(* CODESYS project Base (4).library
   Company: Photara
   DefaultNamespace: Base
   Title: Base
   Placeholder: Base
   Author: Scott Kinder
   Version: 2025.10.17.4

Project tree, tasks and I/O mapping:
  libraries: Tc2_EtherCAT, * (Beckhoff Automation GmbH); Tc2_Standard, * (Beckhoff Automation GmbH); Tc2_System, * (Beckhoff Automation GmbH); Tc2_Utilities, * (Beckhoff Automation GmbH); Tc3_EventLogger, * (Beckhoff Automation GmbH); Tc3_JsonXml, * (Beckhoff Automation GmbH); TcUnit, 1.3.1 (www.tcunit.org)
  Base/
    POUs/
      function block FB_BaseCyclic [ST]: _ConfigurationCyclic, _UpdateStatusEdgeTracking, CyclicLogic, Initialized
      function block FB_BaseStatic [ST]: Busy, Error, ErrorID, Initialize, P_BaseConfiguration, P_BaseStatus, TraceWithSeverity, _FormatLogEntry, _Initialize, _InitializeChildrenDependencies, _InitializeReferences, _SetDependencyConfiguration, RaiseAlarm
    global variables GC_Base
    global variables GPL_Base
    interface I_BaseCyclic: CyclicLogic, Initialized
    interface I_BaseStatic: Busy, Error, ErrorID, Initialize, P_BaseConfiguration, P_BaseStatus, TraceWithSeverity
  Command/
    ITFs/
      interface I_Command: Abort, Cancel, Complete, Execute, InjectConfigurations, P_CommandStatus, Pause, Queue, Reset, Resume, Validate
      interface I_CommandConfiguration: P_CommandConfiguration
      interface I_TestClock: SetElapsedTime
      interface I_Timer: P_ElapsedTime, P_IsElapsed, ResetTimer, StartTimer, StopTimer
    POUs/
      function block FB_Command [ST]: Abort, Cancel, Complete, Execute, InjectConfigurations, P_CommandStatus, Pause, Queue, Reset, Resume, Validate, _Initialize, _InitializeChildrenDependencies, _InitializeReferences, _SetDependencyConfiguration, _AbortCommand, _AbortCommandInterlockLost, _ConfigurationCyclic, _EvaluateConfiguration, _FormatResultString, _FormatStepStateString, _HandleAutoReset, _LogCommand, _MonitorInterlocks, _ProcessStateTransitions, _ResetCommand, _ResolveCommandConfiguration, _ResolveCommandStatus, _ResolvePermIntlkConfiguration, _UpdateComponentStatus, _UpdateStatusEdgeTracking, _ValidateCommand, CyclicLogic, P_CommandConfiguration, P_PermIntlkConfiguration
      function block FB_CommandElapsedTimer [ST]: P_ElapsedTime, P_IsElapsed, ResetTimer, StartTimer, StopTimer, CyclicLogic, InjectConfiguration
  Component/
    GVLs/
      global variables GC_Component
      global variables GPL_Component
    ITFs/
      interface I_ComponentBase: InjectSystemInterfaces, Reset
      interface I_ComponentFull: DequeueCommand, EnqueueCommand, ExecuteCommand, GetIndexByPOUName, HMICommunication, InjectCommandQueue, P_CommandQueue, P_ComponentConfiguration, P_ComponentStatus, ResetAllCommands
    POUs/
      function block FB_Component [ST]: DequeueCommand, EnqueueCommand, ExecuteCommand, GetIndexByPOUName, HMICommunication, InjectCommandQueue, P_CommandQueue, P_ComponentConfiguration, P_ComponentStatus, Reset, ResetAllCommands, _Initialize, _InitializeChildrenDependencies, _InitializeReferences, _SetCommandIndices, _SetCommandPermIntlkConfiguration, FB_Init, InjectCommandConfiguration, InjectPermIntlkConfiguration, InjectSystemInterfaces, _BuildTables, _ClearTempCmdObj, _CommandsCyclic, _ComponentCyclic, _DequeueCommand, _DispatchValid, _EnqueueCommand, _EvaluateCompletionConditions, _InjectCommandConfiguration, _InjectPermIntlkConfiguration, _ObtainAmsNetId, _ProcessCommandQueue, _TryRehashDispatchIndex, _UpdateBusyStatus, _UpdateComponentStatus, CyclicLogic
  Configuration/
    function block FB_CmdPermIntlkConfiguration [ST]: _InitializeReferences, P_CommandConfiguration, P_PermIntlkConfiguration
  ControlMode/
    GVLs/
      global variables GC_ControlMode
      global variables GPL_ControlMode
    ITFs/
      interface I_ControlMode: ChangeMode, P_ControlMode
    POUs/
      function block FB_ControlMode [ST]: ChangeMode, P_ControlMode, _EvaluateCompletionConditions, _UpdateComponentStatus, InjectControlModeCmdPermIntlkConfigurations
  Debounce/
    function block FB_Debounce [ST]: _InitializeReferences, CyclicLogic, P_DebounceConfiguration, P_DebounceStatus, P_RawSignal
    interface I_Debounce: P_DebounceStatus, P_RawSignal
    interface I_DebounceConfiguration: P_DebounceConfiguration
  DUTs/
    Base/
      data type E_DataType
      data type E_HttpStatusCode
      data type E_LinkStatus
      data type ST_BaseConfiguration
      data type ST_BaseStatus
      data type ST_BitSignal
      data type ST_OpStatus
      data type ST_Parameter
      data type ST_PlcSystem
    Command/
      data type E_CommandPriority
      data type E_CommandResult
      data type E_CommandState
      data type ST_CommandConfiguration
      data type ST_CommandStatus
    Component/
      data type E_ComponentTriggerMode
      data type ST_ComponentCommand
      data type ST_ComponentConfiguration
      data type ST_ComponentStatus
    Configuration/
      data type E_ConfigurationResolution
    Debounce/
      data type ST_DebounceConfiguration
      data type ST_DebounceStatus
    EtherCAT/
      data type ST_EtherCATAdsAddr
      data type ST_EtherCATInfoData
      data type ST_EtherCATStatus
      data type ST_EtherCATWcState
    EventHandling/
      data type ST_EventLogHandlerConfiguration
      data type ST_EventLogHandlerStatus
      data type ST_PersistentStorageStatus
    File/
      Structs/
        data type ST_AmsNetId
        data type ST_FileHandlerBaseStatus
        data type ST_FileHandlerConfiguration
        data type ST_FileHandlerCSVConfiguration
        data type ST_FileHandlerCSVStatus
        data type ST_FileHandlerJsonStatus
        data type ST_FileOpStatus
      data type E_FileFormat
    Hash/
      data type ST_HashTableConfiguration
      data type ST_HashTableStatus
    LogTrace/
      data type E_LogTraceWhen
      data type ST_LogBackoffState
      data type ST_LogMetrics
      data type ST_LogTraceConfiguration
      data type ST_LogTraceStatus
      data type ST_LogTraceWhat
    PermIntlk/
      data type E_ModePermIntlk
      data type ST_PermIntlkConfiguration
      data type ST_PermIntlkConfigurationCondition
      data type ST_PermIntlkStatus
      data type ST_PermIntlkStatusCondition
    RingBuffer/
      data type ST_LogEntry
      data type ST_RingBufferCfg
      data type ST_RingBufferStatus
      data type ST_SystimeICmd
      data type ST_SystimeString
    Safety/
      data type ST_SafetyGroupConfiguration
      data type ST_SafetyGroupStatus
    Sequencer/
      data type E_Operation
      data type E_PackMLState
      data type ST_Operation
      data type ST_OperationSequencerConfiguration
      data type ST_OperationSequencerStatus
      data type ST_PackMLSequencerConfiguration
      data type ST_PackMLSequencerStatus
  EventHandling/
    ITFs/
      interface I_LogHandler: AddToEventLog, LogDequeue, MonitorPlcSystem, P_EventLogHandlerStatus
      interface I_LogHandlerConfiguration: P_EventLogHandlerConfiguration
      interface I_PersistentStorage: AddEntry, P_MessagesSentThisScan
      interface I_TraceEvent: AddContext, SetMessage, SetSeverity
    function block FB_EventLogHandler [ST]: CyclicLogic, AddToEventLog, LogDequeue, MonitorPlcSystem, P_EventLogHandlerStatus, P_EventLogHandlerConfiguration, _InitializeChildrenDependencies, _InitializeReferences, _ProcessLogEntry, _UpdatePerformanceMetrics, _UpdateSeverityMetrics, CalculateDynamicRate, HandlePersistenceFailure, UpdateBufferHealthMetrics
    function block FB_PersistentEventLog [ST]: _InitializeChildrenDependencies, _InitializeReferences, AddEntry, P_MessagesSentThisScan
    function block FB_TraceEvent [ST]: AddContext, SetMessage, SetSeverity
    function block FB_UniversalAlarm [ST]: AddContext, Clear, Confirm, Raise, SetMessage, SetSeverity
    function block FB_UniversalMessage [ST]: AddContext, Send, SetMessage, SetSeverity
    global variables GVL_System
  File/
    Function Blocks/
      function block FB_FileHandlerBase [ST]: P_FileHandlerBaseConfiguration, _InitializeReferences, CyclicLogic, P_FileHandlerBaseStatus
      function block FB_FileHandlerJson [ST]: CyclicLogic
    Interfaces/
      interface I_FileHandlerBase: AppendToFileByPointer, CloseFile, CreateFile, DeleteFile, OpenFile, ReadFromFile, RenameFile, WriteFile, P_FileHandlerBaseStatus
      interface I_FileHandlerBaseConfiguration: P_FileHandlerBaseConfiguration
      interface I_FileHandlerCsv: AppendToFileByString, AppendToFileBySystimeString, P_AppendRingBufferStatus, P_FileHandlerCsvStatus
      interface I_FileHandlerJson
    global variables GC_File
    global variables GPL_File
  Functions/
    Numbers/
      function F_IsPowerOfTwo_UINT [ST]
      function F_MapLREAL [ST]
    Strings/
      function F_GetAllButFirstWord [ST]
      function F_GetFirstWordInString [ST]
      function F_GetLastWordInString [ST]
      function F_ReplaceInString [ST]
      function F_TrimString [ST]
    Time/
      function F_DateTimeConvertedAsT_MaxString [ST]
      function F_FILETIME64_TO_LTIME [ST]
      function F_FileTimeToString [ST]
      function F_SystemTimeUtcCorrected [ST]
  Hashing/
    ITFs/
      interface I_HashFunction: Hash
      interface I_HashTableBase: Clear, GetIndex, Insert, P_HashTableStatus
      interface I_HashTableConfiguration: P_HashTableConfiguration
      interface I_HashTableExt: Contains, LoadFactorExceeded, Rehash, Remove
    POUs/
      function block FB_Hash_djb2 [ST]: Hash, P_TP_HashTableStatus
      function block FB_HashTable [ST]: Clear, GetIndex, Insert, P_HashTableStatus, P_HashTableConfiguration, _Initialize, _InitializeChildrenDependencies, _InitializeHashTable, _InitializeReferences, InjectHashFunction
    global variables GPL_HashTable
  PermIntlk/
    GVLs/
      global variables GC_PermIntlk
      global variables GPL_PermIntlk
    ITFs/
      interface I_PermIntlk: Evaluate, InjectPermIntlkConfiguration, P_OK, P_PermIntlkStatus
      interface I_PermIntlkConfiguration: P_PermIntlkConfiguration
    POUs/
      function block FB_PermIntlk [ST]: Evaluate, P_OK, P_PermIntlkConfiguration, _Initialize, _InitializeReferences, _SetElementIndices, _EvaluateConfiguration, _EvaluateOK, _LogMessage, _PermMsgIndexForMessage, _ResolvePermIntlkConfiguration, _ResolvePermIntlkStatus, _ConfigurationCyclic, CyclicLogic, InjectPermIntlkConfiguration, P_PermIntlkStatus, ReinitObjects
      function block FB_PermIntlkCommand [ST]: CyclicLogic, InjectCommandConfiguration
  PRGs/
    program PRG_LOG [ST]
    program PRG_PRETEST [ST]
    program PRG_TEST [ST]
  RingBuffer/
    GVLs/
      global variables GPL_RingBuffer
    ITFs/
      interface I_RingBufferBase: ClearLastRemoved, ClearStatusFlagAdded, ClearStatusFlagPeeked, ClearStatusFlagRead, ClearStatusFlagRemoved, P_ObjectWasAdded, P_ObjectWasPeeked, P_ObjectWasRead, P_ObjectWasRemoved, P_RingBufferStatus, RemoveObject
      interface I_RingBufferICmd: AddObject, P_Buffer, P_LastObjectPeeked, P_LastObjectRead, P_LastObjectRemoved, PeekObject, ReadObject
      interface I_RingBufferKeyString: AddObject, P_Buffer, P_LastObjectPeeked, P_LastObjectRead, P_LastObjectRemoved, PeekObject, ReadObject
      interface I_RingBufferLogEntry: AddObject, P_Buffer, P_LastObjectPeeked, P_LastObjectRead, P_LastObjectRemoved, PeekObject, ReadObject
      interface I_RingBufferString: AddObject, P_Buffer, P_LastObjectPeeked, P_LastObjectRead, P_LastObjectRemoved, PeekObject, ReadObject
      interface I_RingBufferUINT: AddObject, P_Buffer, P_LastObjectPeeked, P_LastObjectRead, P_LastObjectRemoved, PeekObject, ReadObject
    POUs/
      function block FB_RingBufferBase [ST]: _Initialize, _InitializeReferences, UpdateObjectCtInBuffers, P_ObjCountInBuffer, P_ObjectWasAdded, P_ObjectWasPeeked, P_ObjectWasRead, P_ObjectWasRemoved, ClearLastRemoved, IncrementPointer, UpdateRemovePointer, UpdateWritePointer, ClearStatusFlagAdded, ClearStatusFlagPeeked, ClearStatusFlagRead, ClearStatusFlagRemoved, ClearStatusFlags, WrapPointer
      function block FB_RingBufferICmd [ST]: ClearLastRemoved, P_RingBufferStatus, RemoveObject, AddObject, P_Buffer, P_LastObjectPeeked, P_LastObjectRead, P_LastObjectRemoved, PeekObject, ReadObject, UpdateRemovePointer, UpdateWritePointer, _Initialize, ClearBuffer
      function block FB_RingBufferKeyString [ST]: AddObject, ClearLastRemoved, P_LastObjectPeeked, P_LastObjectRead, P_LastObjectRemoved, P_RingBufferStatus, PeekObject, ReadObject, RemoveObject, UpdateRemovePointer, UpdateWritePointer, _Initialize, ClearBuffer, P_Buffer
      function block FB_RingBufferLogEntry [ST]: AddObject, ClearLastRemoved, P_LastObjectPeeked, P_LastObjectRead, P_LastObjectRemoved, P_RingBufferStatus, PeekObject, ReadObject, RemoveObject, UpdateRemovePointer, UpdateWritePointer, _Initialize, ClearBuffer, P_Buffer
      function block FB_RingBufferString [ST]: ClearLastRemoved, P_RingBufferStatus, RemoveObject, AddObject, P_LastObjectPeeked, P_LastObjectRead, P_LastObjectRemoved, PeekObject, ReadObject, UpdateRemovePointer, UpdateWritePointer, _Initialize, ClearBuffer, P_Buffer
      function block FB_RingBufferUINT [ST]: ClearLastRemoved, P_RingBufferStatus, RemoveObject, AddObject, P_LastObjectPeeked, P_LastObjectRead, P_LastObjectRemoved, PeekObject, ReadObject, UpdateRemovePointer, UpdateWritePointer, _Initialize, ClearBuffer, P_Buffer
  Safety/
    GVLs/
      global variables GC_Safety
      global variables GPL_Safety
    function block FB_SafetyDevice [ST]: CyclicLogic
    function block FB_SafetyGroup [ST]: _InitializeReferences, CyclicLogic, P_SafetyGroupConfiguration, P_SafetyGroupStatus, Reset
  Tests/
    FB_CommandConfigured/
      function block FB_CommandConfigured [ST]
    MockFBs/
      function block FB_CommandUnderTest [ST]: SetCommandConfiguration, SetCommandStatus
      function block FB_ComponentDerivative [ST]: P_TP_iSystemPermIntlk, _EvaluateCompletionConditions, _UpdateComponentStatus
      function block FB_ImplBaseCyclic [ST]
      function block FB_ImplBaseStatic [ST]
    TestFunctions/
      function GivenValidCommand [ST]
      function ThenAssertState [ST]
      function WhenExecuteCommand [ST]
    TestInterfaces/
      interface I_CommandUnderTest: SetCommandStatus
    function block FB_BaseCyclicTests [ST]: GivenCyclicCallInitCompleteOK, GivenNoCyclicCallInitCompleteNOK
    function block FB_BaseStaticTests [ST]: GivenInitializationConfigurationReferenceOK, GivenNoInitializationConfigurationReferenceNOK
    function block FB_CommandTestsI [ST]: GivenCommand_WhenCancelCalledIfCommandNotAlreadyDequeuedExpectCommandRemovedFromQueue, GivenCommand_WhenExecuteCalled_ExpectExecutionOccurs, GivenCommand_WhenQueueCalledExpectCommandAddedToQueue, GivenCommand_WhenResetCalled_ExpectStateCleared, GivenCommandInIdleState_WhenCancel_ExpectNoActionTaken, GivenCommandPaused_WhenAbort_ExpectCommandAbortedAndStatusUpdated, GivenCommandQueued_WhenAbort_ExpectCommandAbortedAndStatusUpdated, GivenCommandQueued_WhenCancel_ExpectCommandRemovedFromQueue, GivenComponentReset_WhenResetCalled_ExpectAllCommandStateCleared, TEST_AbortAfterComplete_StatePreservation, TEST_Cancel_FromQueuedState, TEST_Execute_StateMachineProgression, TEST_Execute_TransitionsFromAcceptedToOk, TEST_Reset_ClearsCommandState, TEST_CommandAttemptsExceedRetryCount_ResultTooManyRequests, TEST_CommandTimeout_TriggersReset, TEST_PermIntlkLostDuringBusy_CommandAbortedWithInterlockLost, GivenCommandAlreadyRunning_WhenExecute_ExpectConflictResult, TEST_CommandCompletes_StatusDoneAndBusyCleared, TEST_CompleteState_PreservesAbortedResult, TEST_CompleteState_PreservesTimeoutResult, TEST_CompleteState_SetsOkForSuccessfulCompletion, TEST_Forbidden_ResumeWithoutPermissive_ReturnsForbidden, TEST_OperatorAbort_VsInterlockAbort_DifferentResults, TEST_TerminalResults_ErrorFlagConsistency, TEST_ValidationOK_InterlockDropDuringExecution, TEST_ValidCommand_ExpectExecuted, GivenCommand_WhenCyclicLogicCalled_ExpectStateUpdated, GivenCommand_WhenPauseCalledExpectCommandPauses, GivenCommand_WhenResumeCalledExpectCommandResumes, GivenCommandExecuted_WhenCyclicLogicRuns_ExpectStateProgression, GivenCommandPaused_WhenResume_ExpectCommandResumesExecution, GivenRunningCommand_WhenPause_ExpectCommandTransitionsToPausedState, GivenTimerStarted_WhenCyclicLogicRuns_ExpectElapsedTimeIncreases, GivenTimerStopped_WhenCyclicLogicRuns_ExpectElapsedTimeRemainsConstant, TEST_CyclicLogic_StateMachineProgression, TEST_EdgeTriggered_StateMachineExecution, TEST_PauseResume_StateTransitions, TEST_StepState_TransitionsAndValidation, GivenCommand_WhenValidateCalled_ExpectPermissiveOK, GivenCommand_WhenValidateCalled_ExpectValidationResultMatchesConfiguration, GivenCommandInvalid_WhenValidateCalled_ExpectFalse, GivenCommandValidated_WhenValidateCalled_ExpectTrue, GivenInjectedConfigurationsValid_WhenInjectConfigurations_ExpectInterfacesStoredAndInitialized, GivenInvalidConfiguration_WhenInjectConfigurationCalled_ExpectInitializationFailure, GivenInvalidConfigurations_WhenInjectConfigurations_ExpectInitializationFailure, GivenValidConfiguration_WhenInjectConfigurationCalled_ExpectConfigurationStored, TEST_ComponentBusyDuringValidation_ResultConflict, TEST_InjectConfigurations_StoresInterfacesProperly, TEST_InterfaceInjectionConfigurationResolution, TEST_PermissiveFalseDuringValidation_ResultForbidden, TEST_Validate_ReturnsProperResultBasedOnPermissives, TEST_Validate_WithContinuousEvaluation
    function block FB_CommandTestsII [ST]: TEST_Abort_AfterComplete_IgnoredWithWarning, TEST_Abort_WhenIdleQueued_SetsResultAbortedAndRemovesFromQueue, TEST_Cancel_WhenBusy_RejectedWithWarning_NoStateChange, TEST_Execute_HappyPath_TransitionsToMonitorAndCompletesOk, TEST_Execute_WhenPermissiveMissing_ReturnsForbidden, TEST_RetryCount_IncrementOnExecutionStartOnly, TEST_TimeoutAndInterlockLost_SameCycle_PrioritizeInterlockLost, TEST_Complete_Error_PersistsUntilReset, TEST_Complete_Ok_AutoResetsNextCycle, TEST_SystematicStateValidation_IdleStates, TEST_SystematicStateValidation_TerminalStates, TEST_Config_FallbackToLocal_WhenInjectedInvalid, TEST_Config_RecoveryToInjected_WhenValidAgain, TEST_Execute_ValidatesBeforeAccepting, TEST_RuntimeCommandConfigLoss_InjectedRefsInvalidatedDuringExecution, TEST_RuntimeCommandConfigRecovery_ValidRefsRestoredDuringExecution, TEST_AbortDuringCompletionWait, TEST_CompletionCallbackToSequencer, TEST_CompletionConditionEvaluation, TEST_CompletionWithInterlockDrop, TEST_DiscreteCompletionCondition, TEST_DynamicCompletionConditionUpdate, TEST_FastCompletionInOneScan, TEST_MotionCompletionCondition, TEST_OperationToCommandTranslation, TEST_RecipeManagerProvidesCommandConfig, TEST_TimeBasedCompletionCondition
    function block FB_CommandTestsIII [ST]: TEST_MethodEnablement_BusyState_ShouldAllowAbortRejectExecute, TEST_MethodEnablement_DoneState_ShouldAllowResetRejectExecute, TEST_MethodEnablement_IdleWithInterlockOK_ShouldAllowExecute, TEST_MethodEnablement_IdleWithoutInterlockOK_ShouldRejectExecute, TEST_InterlockInvalidConfigurationDuringValidation_ReturnsBadRequest, TEST_InterlockReferenceLostDuringExecution_FallsBackOrAborts, TEST_InterlockDrop_AbortsCommandWhenConfigured, TEST_InterlockDrop_FromMonitorState_CommandAborted, TEST_InterlockLost_ComprehensiveStateTransitions, TEST_InterlockLost_FromExecuteState, TEST_InterlockLost_SetsCorrectResult, TEST_TimerCompletionTime_SetOnCommandComplete, TEST_TimerIntegration_WithCommandStateMachine, TEST_TimerPauseResume_ElapsedTimeAccuracy, TEST_TimerStopsOnCommandComplete_NotTimeout, TEST_TimerTriggerTime_SetOnCommandStart
    function block FB_CommandTestsIV [ST]: TEST_Abort_ErrorClassification, TEST_Cancel_RemovesCommandFromQueue, TEST_Cancel_SetsCommandStatusToCancelled, TEST_Cancel_SetsResultToCancelled, TEST_BadRequest_InterlockMisconfigured_ReturnsBadRequest, TEST_BusyCommandElapsedTimeEqualsTimeout_CommandAborted, TEST_AcceptedCommand_WhenExecuted_ResultBecomesOk, TEST_Command_LocalReferences_InitializedProperly, TEST_Command_MissingConfigInterface_FallbackToLocal, TEST_Command_PermIntlkChild_Initialized, TEST_CommandStatus_ConfigRef_PointsToConfiguration
    function block FB_CommandTestsV [ST]: TEST_ConfigurationResolution_HandlesValidAndInvalidInterfaces, TEST_ResultPersistence_TerminalStates, TEST_AbortDuringCompletionWait, TEST_CompletionCallbackToSequencer
    function block FB_CommandTestsVI [ST]: TEST_DynamicCompletionConditionUpdate, TEST_PauseResumeWithCompletionCondition
    function block FB_CommandTestsVII [ST]: TEST_Busy_FalseToTrue_OnStart_TrueToFalse_OnComplete
    function block FB_ComponentTests [ST]: TEST_Component_ChildrenDependencies_Initialized, TEST_Component_InitComplete_SetAfterInitialize, TEST_Component_Initialize_OnlyCalledOnce, TEST_Component_MissingCommandInterface_HandlesGracefully, TEST_Component_MissingPermIntlkInterface_HandlesGracefully, TEST_Component_QueryInterface_ValidatesTypes, TEST_ComponentConfiguration_BaseConfiguration_ReferenceValid, TEST_ComponentStatus_BaseStatus_ReferenceValid, GivenAbortInvokedDuringValidation_CommandNeverEnqueuedOrExecuted, GivenBusyCommandElapsedTimeEqualsTimeout_CommandAborted, GivenCommandBusyAndInterlockLostWithAbortOnInterlockDrop_AbortFires, GivenCommandBusyAndInterlockLostWithoutAbortOnInterlockDrop_CommandContinues, GivenCommandBusyAndInterlockStaysOk_NoAbortOccurs, GivenComponentBusyDuringValidation_ResultConflict, GivenIndeterminantCommandDequeuedButPermissiveDropsBeforeExecute_ResultForbiddenNotOk, GivenInterlockNotInitComplete_CommandValidationFailsForbidden, GivenPermIntlkAllRequiredItemsTrue_EvaluateOKReturnsTrue, GivenPermIntlkInitNotComplete_EvaluateOKReturnsFalse, GivenPermIntlkLostDuringBusy_WhenAbortOnInterlockDropFalse_CommandContinues, GivenPermIntlkOptionalItemFalse_EvaluateOKReturnsTrue, GivenPermIntlkRequiredItemFalse_EvaluateOKReturnsFalse, GivenPermissiveFalseDuringValidation_ResultForbidden, GivenResetCalledOnBusyCommand_ResultsInAbortThenNone, GivenAbortOnBusyCommand_LastCommandStatusUpdated, GivenAcceptedCommand_WhenExecuted_ResultBecomesOk, GivenBusyCommandElapsedTimeMeetsTimeout_WhenCmdTryCountEqualsConfiguredRetryCount_CommandIsAbortedAndMarkedTooManyRequests, GivenBusyCommandElapsedTimeMeetsTimeout_WhenCmdTryCountIsLessThanConfiguredRetryCount_CommandIsAbortedAndRequeued, GivenBusyCommandTimeoutBeforeRetry_RetryEnqueued, GivenBusyFlagTrueForAcceptedCommand_TurnsFalseOnlyAfterOkOrAbort, GivenCommandAborted_LastCommandStatusReflectsAbort, GivenCommandAborted_LastCommandStatusShowsAbortedUntilNextCommandRuns, GivenCommandAbortedThenReEnqueued_CommandTryCountResetsToPreviousPlusOne, GivenCommandAttemptsExceedRetryCount_ResultTooManyRequests, GivenCommandCompletes_CommandStatusDoneAndBusyCleared, GivenCommandExecutes_LastCommandStatusUpdatedToCurrentCommand, GivenCommandIsBusy_WhenNextCommandQueued_SecondCommandRemainsInQueue, GivenCommandPreempted_LastCommandStatusReflectsNewCommand, GivenCommandRetriesPastMaxAttempts_ResultTooManyRequests, GivenCommandTimesOutOnce_ResultRequestTimeout, GivenCreatedCommand_WhenDequeued_ResultIsAccepted, GivenEqualPriorityCommandQueued_ExistingBusyCommandNotAborted, GivenEqualPriorityCommandQueued_RunningCommandContinues, GivenExecutionTypeImmediateReturn_WhenDequeued_ResultTransitionsDirectlyToOkWithoutBusy, GivenExecutionTypeIndeterminant_WhenCommandValidated_ResultCreatedThenAcceptedThenBusy, GivenHigherPriorityCommandQueued_AbortsLowerPriorityRunningCommand, GivenIndeterminantCommandDequeued_ComponentBusyFlagSetTrueUntilCompletion, GivenNewCommandDequeued_LastCommandStatusSwitchesFromOldToNew, GivenNoBusyCommands_ComponentStatusBusyFalse, GivenOneBusyCommand_ComponentStatusBusyTrue, GivenQueuedCommand_ComponentStatusBusyFalseUntilExecution, GivenThatCommandIsBusyQueueNextCommand, GivenTimeoutZero_DisablesTimeoutLogic, GivenUseCommandPriorityFalse_NoPreemptionRegardlessOfPriority, GivenValidatedCommand_WhenEnqueued_ResultIsCreated, GivenAbortCalledTwice_IdempotentStateUnchangedSecondTime, GivenAllCommandInterfacesMissing_ComponentCyclicLogicDoesNotCrash, GivenChangingCommandConfigurationDuringBusyCommand_NoPointerCorruptionOrUnexpectedAbort, GivenCommandCancelledBeforeDequeued_ResultChangesToAbortedWithoutExecution, GivenCommandExecutesLongerThanConfiguredTimeoutButFinishes_SuccessfulCompletionOverridesTimeoutAbort, GivenCommandMarkedTooManyRequestsAndReset_AllowedToRequeueWithTryCountZero, GivenCommandResetWhileQueued_ResultChangesFromCreatedToNone, GivenComponentReset_AllChildReferencesRemainValid, GivenComponentReset_LastCommandStatusClearedOrResetAsConfigured, GivenComponentRestartWhileCommandsQueued_PendingQueueClearedOrRecoveredGracefully, GivenExceededRetryLimit_CommandResultTooManyRequestsAndNoRequeue, GivenInterlockNotConfigured_ValidationIgnoresPermIntlkPointer, GivenInvalidCmdIndex_ResultUnprocessableEntity, GivenInvalidCommand_ExpectError, GivenInvalidCommandIndexGreaterThanUpperBound_ExecuteCommandReturnsUnprocessable, GivenLastCommandStatusUpdatedOnAbortThenOnNextExecute_NoStalePointer, GivenMissingCommandInterface_ResultUnprocessableEntity, GivenMissingConfigInterface_ResultUnprocessableEntity, GivenMissingPermIntlkInterface_ResultUnprocessableEntity, GivenNullComponentReferenceInCommand_ValidationAndExecutionNoOpsWithoutError, GivenNullPermIntlkPointer_WhenPermIntlkConfiguredFalse_ValidationPasses, GivenNullRingBufferPointer_WhenComponentExecutesValidation_NoNullPointerAccess, GivenPermIntlkNotLinkedToCommand_NoEvaluationOccursDuringCyclic, GivenPriorityOverflow_NoRuntimeException, GivenPriorityOverflowThenWrap_NoSchedulerCrash, GivenResetCalledOnCompletedCommand_StatusResetToNone, GivenRetryLimitExceededDuringValidation_ResultTooManyRequests, GivenRingBufferFull_WhenNewCommandEnqueued_ResultHeaderTooLarge, GivenRingBufferNotConfigured_EnqueueLogsFailure, GivenRingBufferWrapAround_NoCommandLostDuringContinuousEnqueueDequeue, GivenUnexpectedExceptionThrownInCommandExecute_ResultInternalServerErrorSetAndSystemContinues, GivenValidInterfaces_WhenComponentIdle_CommandValidatesContinues, GivenActiveCommand_CyclicLogicAlwaysCalledEachScan, GivenCommandAttemptedWithRetryCountEqualToConfiguredRetryCount_NoFurtherRetries, GivenCommandAttemptedWithRetryCountLessThanConfiguredRetryCount_RetryAllowed, GivenExecutionTypeImmediateReturn_WhenCommandValidated_ResultCreatedAndBusyNeverTrue, GivenExecutionTypeImmediateReturn_WhenTimeoutPeriodElapsed_NoTimeoutOccurs, GivenExecutionTypeIndeterminant_WhenBusyAndTimeoutExceeded_CommandRetriesOrFailsPerRetryCount, GivenHighPriorityCommandInsertedLate_PreemptsLowerPriorityBeforeExecutionStarts, GivenImmediateDequeueDisabled_CommandWaitsForNextCyclicExecution, GivenImmediateDequeueEnabled_CommandValidatedAndExecutedSameScan, GivenImmediateReturnAndIndeterminantInSameQueue_OrderOfCompletionReflectsQueueOrder, GivenImmediateReturnCommandDequeuedWhileComponentIdle_CompletesWithoutAffectingBusyFlag, GivenImmediateReturnCommandQueuedDuringBusyCommand_QueuesBehindButDoesNotPreempt, GivenImmediateReturnCommandQueuedWhileComponentBusy_CompletesInSameCycleAfterBusyClears, GivenImmediateReturnCommandWithAbortOnInterlockDropTrue_InterlockDropHasNoEffect, GivenImmediateReturnCommandWithZeroTimeout_DoesNotError, GivenInactiveCommand_CyclicLogicNotCalledToSaveCPU, GivenIndeterminantCommandWithZeroTimeout_TimesOutNextScan, GivenLowerPriorityCommandQueued_ReEnqueuedUntilRunningCommandFinishes, GivenMultipleCommandsHitTimeoutSimultaneously_AbortAndRetryOccursForEachCommandIndependently, GivenMultipleCommandsSamePriorityStartedSequentially_OnlyOneBusy, GivenMultipleImmediateReturnCommandsQueuedTogether_AllCompleteWithinSameScan, GivenMultipleLowerPriorityCommandsQueuedInBurst_ExecutionOrderPreservedFIFO, GivenNewHighPriorityCommandArrivesWhileBusy_OldCommandAbortedNewExecutes, GivenNoNewCommandsForNScans_LastCommandStatusRemainsUnchanged, GivenPermIntlkConfiguredAsFalse_CommandChecksOnlyAtStart_NoMidRunAbort, GivenPermIntlkConfiguredAsFalse_InterlockIgnoredDuringExecution, GivenPermIntlkEvaluateCalledEveryCycleWhileBusy_ToggleDetectedWithinOneScan, GivenPermIntlkFlappingRapidlyDuringBusyCommand_CommandAbortsOnlyAfterPersistentDrop, GivenPermIntlkFlapsLongerThanDebounce_AbortTriggered, GivenPermIntlkFlapsShorterThanDebounce_NoAbortTriggered, GivenPermIntlkTransitionFromFalseToTrue_EvaluateOKChangesAfterNextEvaluate, GivenPermissiveDropsForOneCycle_CommandNotAbortedUnlessDropPersists, GivenQueueContainsMixedPriorities_CorrectOrderRespectedEvenAfterReEnqueue, GivenReEnqueuedAfterTimeout_NewCommandResultIsCreated, GivenRetryCommandFinishesSuccessfully_PreviousTimeoutDoesNotBlockFutureEnqueue, GivenRetryTriggered_CommandReenqueuedAsNewQueueEntryWithIncrementedTryCount, GivenTimeoutAbort_LastCommandStatusReflectsRequestTimeoutReason, GivenTimeoutAfterFinalRetry_CommandStatusForeverTooManyRequestsUntilReset, GivenTimeoutAndRetryPolicyDisabled_CommandResetImmediately, GivenTimeoutRetryPath_ComponentBusyFlagClearsDuringAbortAndRemainsFalseUntilDequeuedAgain, GivenTimeoutValueShorterThanScanTime_CommandStillRetriesProperly, GivenTimeoutWithRetriesRemaining_CommandStatusFlipsAbortedThenCreatedWithinSameScan
    function block FB_DebounceTests [ST]: GivenAlternatingNoise_WhenBelowTONAndTOF_ExpectOutputStable, GivenDebounceActive_WhenOutputFalse_ExpectStatusConsistent, GivenDebounceActive_WhenOutputTrue_ExpectStatusConsistent, GivenInputHigh_WhenHeldLongerThanTON_ExpectOutputTrue, GivenInputHigh_WhenReleasedBeforeTON_ExpectOutputFalse, GivenInputHigh_WhenTONExpired_ExpectQRiseTrue, GivenInputHigh_WhenTONNotExpired_ExpectQRiseFalse, GivenInputLow_WhenHeldLongerThanTOF_ExpectOutputFalse, GivenInputLow_WhenReleasedBeforeTOF_ExpectOutputTrue, GivenInputLow_WhenTOFExpired_ExpectQFallTrue, GivenInputLow_WhenTOFNotExpired_ExpectQFallFalse, GivenMultipleCycles_WhenInputStable_ExpectNoRepeatedQRiseOrQFall, GivenShortHighPulse_WhenShorterThanTON_ExpectNoQRise, GivenShortLowPulse_WhenShorterThanTOF_ExpectNoQFall, GivenSimulationDisabled_WhenDebounceRuns_ExpectHardwareSignalUsed, GivenSimulationEnabled_WhenDebounceRuns_ExpectSimulatedSignalUsed, GivenStableHigh_WhenNoTransition_ExpectNoQRise, GivenStableLow_WhenNoTransition_ExpectNoQFall, GivenTONAndTOFZero_WhenDebounceRuns_ExpectImmediateOutputChange, GivenTransitionHighToLow_WhenDebounced_ExpectQFallTrue, GivenTransitionLowToHigh_WhenDebounced_ExpectQRiseTrue, GivenValidConfiguration_WhenInitialized_ExpectOutputFalse
    function block FB_FileHandlerCsvTests [ST]: TEST_CloseFileCommandDispatch
    function block FB_HashTableTests [ST]: GivenBadCapacity_ExpectRefusalToInitialize, GivenEdgeCaseKeys_ExpectProperHandling, GivenEmptyTable_WhenLookup_ExpectNotFound, GivenExistingKey_WhenInsertWithNewValue_ExpectValueUpdated, GivenFullTable_ExpectGracefulHandling, GivenHashCalledTwice_ExpectSameOutput, GivenInsertThenLookup_ExpectIndexReturned, GivenKeysWithCollision_ExpectBothRetrievable, GivenMixedOperations_ExpectConsistentCount, GivenPopulatedTable_WhenClear_ExpectEmptyTable
    function block FB_InterfaceResolutionTests [ST]: GivenActuatorWithInjectedInterfacesExpectAllInterfacesValid, GivenCommandStatusExpectAllResolvedOrInjected, FB_Init
    function block FB_LogTests [ST]: GivenAllTasksMonitored_WhenMonitorPlcSystemRuns_ExpectUtilizationPercentagesCalculated, GivenBufferHasEntries_WhenDequeueRuns_ExpectEntriesForwarded, GivenBufferNearCapacity_WhenDequeueRuns_ExpectRateIncreased, GivenBufferOverflow_WhenUpdateBufferHealthMetrics_ExpectOverflowCountIncremented, GivenEmergencyFill_WhenDequeueRuns_ExpectMaxRateCappedAt200, GivenEmptyBuffer_WhenLogDequeueCalled_ExpectNoErrors, GivenFailureOnPersistence_WhenAddToEventLog_ExpectFalseReturned, GivenFirstCycle_WhenProgramRuns_ExpectInitializationComplete, GivenHighLoad_WhenDequeueRuns_ExpectRateReduced, GivenLogProcessing_WhenUpdatePerformanceMetrics_ExpectThroughputCalculated, GivenMaxBackoffReached_WhenHandleFailureCalled_ExpectNoFurtherIncrease, GivenMultipleCycles_WhenUpdatePerformanceMetrics_ExpectRollingAverageUpdated, GivenNormalLoad_WhenUpdateBufferHealthMetrics_ExpectAccurateUtilization, GivenNormalOperation_WhenLogDequeueCalled_ExpectEntriesProcessed, GivenProcessing_WhenUpdateSeverityMetrics_ExpectSeverityCountersCorrect, GivenQueueOverflow_WhenEnqueueCalled_ExpectOldestEntriesDroppedGracefully, GivenRepeatedPersistenceFailures_WhenHandleFailureCalled_ExpectExponentialBackoffApplied, GivenSuccessfulPersistence_WhenAddToEventLog_ExpectTrueReturned, GivenTaskCycleExceed_WhenMonitorPlcSystemRuns_ExpectCriticalEventLogged, GivenTaskWithinLimits_WhenMonitorPlcSystemRuns_ExpectNoViolationLogged, GivenBufferFull_WhenNewCriticalEntryArrives_ExpectSpaceReservedForCritical, GivenBufferNearFull_WhenCriticalAndDebugEntriesEnqueued_ExpectCriticalEntriesPreserved, GivenExtendedPersistenceFailure_WhenRecovered_ExpectRateGraduallyRestored, GivenHighJitter_WhenMonitoringTaskUtilization_ExpectCorrectHealthScoreLogged, GivenMaxDequeueLoad_WhenCycleRuns_ExpectTaskNotToExceed50ms, GivenOverflowCondition_WhenMetricsUpdated_ExpectDroppedCountAccurate, GivenPersistenceBlocked_WhenHandleFailureRuns_ExpectProcessingSuspendedUntilTimeout, GivenPersistenceThrowsException_WhenAddToEventLog_ExpectSafeRecovery, GivenProcessingAcrossAllSeverities_WhenMetricsUpdated_ExpectAccurateSeverityDistribution, GivenRestart_WhenLoggerResumes_ExpectMetricsResetAndSafeStartup, GivenBackoffTimerActive_WhenNextCycleRuns_ExpectNoPrematureRetries, GivenBufferAtMaxCapacity_WhenFloodedWithEntries_ExpectGracefulDegradation, GivenBufferOverflow_WhenRecovered_ExpectMetricsReflectCorrectDropCounts, GivenCycleExceeds_WhenDetected_ExpectHealthScoreReducedAndViolationLogged, GivenHeavyOSLoad_WhenPersistenceSlows_ExpectLoggerTaskStillMeetsCycleTime, GivenMaxDequeueRate_WhenCycleRuns_ExpectCycleTimeWithin50msBudget, GivenMixedSeverityFlood_WhenProcessing_ExpectLatencyForCriticalEntriesLow, GivenMultipleTasksMonitored_WhenSystemStable_ExpectUtilizationReportedAccurately, GivenPersistenceThrowsUnhandledException_WhenCaught_ExpectNoTaskCrash, GivenRepeatedPersistenceFailure_WhenRecovered_ExpectRateRestoredToNormal, GivenSeverityMix_WhenProcessing_ExpectSeverityDistributionAccurate, GivenSustainedHighThroughput_WhenRunningFor10Minutes_ExpectNoMemoryLeakOrCycleExceed
    function block FB_PermIntlkTests [ST]: GivenAllConditionsFalse_WhenModeAllConditions_ExpectPermIntlkNotOK, GivenAllConditionsFalse_WhenModeAnyConditions_ExpectPermIntlkNotOK, GivenAllConditionsTrue_WhenModeAllConditions_ExpectPermIntlkOK, GivenAllConditionsTrue_WhenModeAnyConditions_ExpectPermIntlkOK, GivenConfigurationInjection_ExpectProperResolution, GivenLocalFallbackConfiguration_ExpectProperOperation, GivenNoConfiguration_ExpectDefaultTrueBehavior, GivenOneConditionFalse_WhenModeAllConditions_ExpectPermIntlkNotOK, GivenOneConditionTrue_WhenModeAnyConditions_ExpectPermIntlkOK, GivenUnconfiguredConditions_ExpectDefaultTrueBehavior, TEST_ConfigResolution_RecoversToInjected_WhenRefsValidAgain, TEST_ConfigResolution_SwitchesInjectedToLocal_WhenRefsInvalid, TEST_ConfiguredFlag_EmptyDescription_TreatedAsUnconfigured, TEST_Initialize_Twice_IsIdempotent_NoDuplicateSideEffects, TEST_Permissive_Fall_LogsInterlockLost_Once, TEST_Permissive_Rise_LogsPermissiveOK_Once, TEST_Permissive_Toggle_NoLogSpam, TEST_ReinitObjects_ClearsLocalConfig_AndSetsP_OK_TRUE, TEST_RuntimeConfigLoss_InjectedRefsInvalidatedDuringExecution, TEST_RuntimeConfigRecovery_ValidRefsRestoredDuringExecution, TEST_SetElementIndices_AssignsMissingIndices_ForInjectedConfig
    function block FB_RingBufferLoggerTests [ST]: GivenAdd3ObjectExpect3ObjectToBeAdded, GivenAdd3Remove3ExpectFifoOrder, GivenAddAndRemoveAlternateExpectFIFOOrder, GivenAddExactCapacityThenRemoveAllExpectFIFO, GivenAddExpectCorrectByteCount, GivenAddMaxUDINTObjectsExpectGracefulHandling, GivenAddMoreThanCapacityExpectCorrectGlobalCounter, GivenAddMoreThanDoubleCapacityThenReadAllExpectOnlyRecent, GivenAddNullString_ExpectHandledGracefully, GivenAddObjectExpectStatusFlagsUpdateCorrectly, GivenAddObjectLength10ExpectObjectToBeAdded, GivenAddObjectLength20ExpectObjectToBeAdded, GivenAddObjectLength40ExpectObjectToBeAdded, GivenAddObjectLength80ExpectObjectToBeAdded, GivenAddRemoveExpectFlagsSet, GivenAddRemoveOneObjectExpectSameObjectBack, GivenAddThenClearLastRemovedExpectEmptyFlag, GivenAddThenQueryPointerConsistency, GivenAddThenReadExpectSameObject, GivenAddThenRemoveExpectCorrectCounters, GivenAddWhileRemoveInProgressExpectNoCorruption, GivenAddWithInvalidRefExpectNoWrite, GivenClearBufferExpectObjectCountZero, GivenClearCalledExpectAllStatsReset, GivenCopyMemAreaValidInputExpectDataCopiedCorrectly, GivenEmptyBufferExpectPeekReturnsDefault, GivenFillBufferExpectIsFullTrue, GivenFullBufferAddOneExpectOverwriteOldest, GivenInitExpectDefaultPointerAndState, GivenLargeStringExpectTruncationOrError, GivenMultipleAddInSingleCycleExpectAllStored, GivenMultipleAddsSameCycleExpectAllStored, GivenMultipleObjectsExpectPeekAlwaysReturnsFirst, GivenNullRefInputExpectGracefulHandling, GivenOneObjectAddedExpectPeekReturnsIt, GivenOversizedObject_WhenAdded_ExpectNoAdjacentMemoryCorruption, GivenOversizedObjectExpectPartialWriteOrError, GivenOverwrite_WhenOccurs_ExpectDropCounterIncremented, GivenOverwriteExpectFlagSet, GivenOverwriteOccursExpectOnlyRecentN, GivenOverwriteThenReadExpectMostRecent, GivenOverwriteThenRemoveExpectOverwriteCleared, GivenPeekAndReadExpectFlagsSet, GivenPeekThenClearPeekedFlagExpectReset, GivenRapidAddRemoveInLoopExpectCorrectFinalCount, GivenReadFromEmptyExpectNoCrashOrInvalid, GivenReadThenClearStatusExpectFlagsReset, GivenReadThenRemoveExpectCorrectFlagsAndCounts, GivenRemoveBeyondCapacity_ExpectSafeReset, GivenRemoveFromEmptyExpectError, GivenRemoveObjectExpectLastRemovedMatchesExpected, GivenRemoveOnEmptyExpectNoCrash, GivenRemovePointerWrapsAroundExpectValidRead, GivenRemoveThenReadExpectNoNewData, GivenUpdateRemovePointerBoundaryExpectCorrectWrap, GivenUpdateWritePointerBoundaryExpectCorrectWrap, GivenWrapAroundManyTimes_ExpectCountersStable, GivenWrapAroundReadPointerExpectCorrectRead, GivenWrapAroundWriteExpectValidRead, GivenWritePointerWrapsAroundExpectValidOverwrite, GivenZeroCapacityBufferExpectNoWrite, Test_BufferStatus_Add4Remove2, Test_BufferStatus_AfterAddAndRemove
    function block FB_RingBufferTests [ST]: GivenAdd3ObjectExpect3ObjectToBeAdded, GivenAdd3Remove3ExpectFifoOrder, GivenAddAndRemoveAlternateExpectFIFOOrder, GivenAddExactCapacityThenRemoveAllExpectFIFO, GivenAddExpectCorrectByteCount, GivenAddMaxUDINTObjectsExpectGracefulHandling, GivenAddMoreThanCapacityExpectCorrectGlobalCounter, GivenAddMoreThanDoubleCapacityThenReadAllExpectOnlyRecent, GivenAddObjectExpectStatusFlagsUpdateCorrectly, GivenAddObjectLength10ExpectObjectToBeAdded, GivenAddObjectLength20ExpectObjectToBeAdded, GivenAddObjectLength40ExpectObjectToBeAdded, GivenAddObjectLength80ExpectObjectToBeAdded, GivenAddRemoveExpectFlagsSet, GivenAddRemoveOneObjectExpectSameObjectBack, GivenAddThenClearLastRemovedExpectEmptyFlag, GivenAddThenQueryPointerConsistency, GivenAddThenReadExpectSameObject, GivenAddThenRemoveExpectCorrectCounters, GivenAddWhileRemoveInProgressExpectNoCorruption, GivenAddWithInvalidRefExpectNoWrite, GivenClearBufferExpectObjectCountZero, GivenClearCalledExpectAllStatsReset, GivenCopyMemAreaValidInputExpectDataCopiedCorrectly, GivenEmptyBufferExpectPeekReturnsDefault, GivenFillBufferExpectIsFullTrue, GivenFullBufferAddOneExpectOverwriteOldest, GivenInitExpectDefaultPointerAndState, GivenLargeStringExpectTruncationOrError, GivenMultipleAddInSingleCycleExpectAllStored, GivenMultipleAddsSameCycleExpectAllStored, GivenMultipleObjectsExpectPeekAlwaysReturnsFirst, GivenNullRefInputExpectGracefulHandling, GivenOneObjectAddedExpectPeekReturnsIt, GivenOversizedObjectExpectPartialWriteOrError, GivenOverwriteExpectFlagSet, GivenOverwriteOccursExpectOnlyRecentN, GivenOverwriteThenReadExpectMostRecent, GivenOverwriteThenRemoveExpectOverwriteCleared, GivenPeekAndReadExpectFlagsSet, GivenPeekThenClearPeekedFlagExpectReset, GivenRapidAddRemoveInLoopExpectCorrectFinalCount, GivenReadFromEmptyExpectNoCrashOrInvalid, GivenReadThenClearStatusExpectFlagsReset, GivenReadThenRemoveExpectCorrectFlagsAndCounts, GivenRemoveFromEmptyExpectError, GivenRemoveObjectExpectLastRemovedMatchesExpected, GivenRemoveOnEmptyExpectNoCrash, GivenRemovePointerWrapsAroundExpectValidRead, GivenRemoveThenReadExpectNoNewData, GivenUpdateRemovePointerBoundaryExpectCorrectWrap, GivenUpdateWritePointerBoundaryExpectCorrectWrap, GivenWrapAroundReadPointerExpectCorrectRead, GivenWrapAroundWriteExpectValidRead, GivenWritePointerWrapsAroundExpectValidOverwrite, GivenZeroCapacityBufferExpectNoWrite, Test_BufferStatus_Add4Remove2, Test_BufferStatus_AfterAddAndRemove
    function block FB_StringParsingFunctionTests [ST]: TEST_F_GetLeadingWord, TEST_F_StringAfterLastDot, TEST_ReplaceInString
    global variables GC_Test
*)

// DUTs/Base/E_DataType
{attribute 'qualified_only' := ''}
{attribute 'to_string' := ''}
TYPE E_DataType :
(
	ERROR,
	BOOL_TYPE,
	BIT_TYPE,
	BYTE_TYPE,
	WORD_TYPE,
	DWORD_TYPE,
	LWORD_TYPE,
	REAL_TYPE,
	LREAL_TYPE,
	USINT_TYPE,
	UINT_TYPE,
	UDINT_TYPE,
	ULINT_TYPE,
	SINT_TYPE,
	INT_TYPE,
	DINT_TYPE,
	LINT_TYPE,
	STRING_TYPE,
	WSTRING_TYPE,
	CAN_TYPE,
	POINTER_TO_AXIS_TYPE,
	MAX_ENUM
);
END_TYPE

// DUTs/Base/E_HttpStatusCode
{attribute 'qualified_only'}
{attribute 'to_string'}
TYPE E_HttpStatusCode :
(
    ContinueRequest     := 100,
    SwitchingProtocol   := 101,
    Processing          := 102,
    Ok                  := 200,
    Created             := 201,
    Accepted            := 202,
    MultipleChoice      := 300,
    MovedPermanently    := 301,
    Found               := 302,
	TempRedirect		:= 307,
    BadRequest          := 400,
    Unauthorized        := 401,
    Forbidden           := 403,
    NotFound            := 404,
    MethodNotAllowed    := 405,
	NotAcceptable		:= 406,
	ProxyAuthRequire	:= 407,
	RequestTimeout		:= 408,
	Conflict			:= 409,
	PayloadTooLarge		:= 413,
	ImATeapot			:= 418,
	EnhanceYourCalm		:= 420,
	UnprocessableEntity	:= 422,
	TooManyRequests		:= 429,
	HeaderTooLarge		:= 431,
	InvalidToken		:= 498,
	TokenRequired		:= 499,
    InternalServerError := 500,
    NotImplemented      := 501,
	BadGateway			:= 502,
	ServiceUnavailable	:= 503,
	GatewayTimeout		:= 504
) UDINT := NotImplemented;
END_TYPE

// DUTs/Base/E_LinkStatus
{attribute 'qualified_only'}
{attribute 'strict'}
{attribute 'to_string'}
TYPE E_LinkStatus :
(
	NotLinked := 0, 
	Linked	:= 1
) := NotLinked;
END_TYPE

// DUTs/Base/ST_BaseConfiguration
TYPE ST_BaseConfiguration :
STRUCT
	InstancePath				: REFERENCE TO STRING;
	LogTraceConfiguration		: ST_LogTraceConfiguration;
	UseLocalConfig				: BOOL; //FALSE ; Use GPL (Global Param List)
	InSimulation				: BOOL := FALSE; // Allow Tests to trigger this BOOL to write status directly, to put the function block in a particular state for testing
END_STRUCT
END_TYPE

// DUTs/Base/ST_BaseStatus
TYPE ST_BaseStatus :
STRUCT
	Done				: BOOL;
	Busy 				: BOOL;
	Error				: BOOL;
	ErrorID				: UDINT;
	Initialized			: BOOL;
	Enabled				: BOOL := TRUE;
	Simulation			: BOOL;
	LogEntry			: ST_LogEntry;
	LogTraceStatus		: ST_LogTraceStatus;
END_STRUCT
END_TYPE

// DUTs/Base/ST_BitSignal
TYPE ST_BitSignal :
STRUCT
	Ptr 		: POINTER TO BYTE; // Assign Raw IO signal to this pointer to BYTE (PtrSignal := ADR(Signal))
	BitNo		: SINT; //Set in Final Protocol library's FB_INIT, IF Trigger %I*/%Q* is BOOL Bit Number is 0
	MutexLock	: BOOL; //Set for multiple thread accessing the same byte area. Set priority.
	Priority	: SINT; //Set only for multithreading access control with MutexLock (1 to 8 priority for 8 bits in a byte)
	Active		: BOOL; //Signal stored for when bit is set high for outputs OR actively monitoring for inputs
END_STRUCT
END_TYPE

// DUTs/Base/ST_OpStatus
TYPE ST_OpStatus : 
STRUCT
	Operating 	: BOOL 	:= TRUE;
	Description : STRING := 'Not Configured; overwrite in _OpStatus';
END_STRUCT
END_TYPE

// DUTs/Base/ST_Parameter
TYPE ST_Parameter :
STRUCT
	ParameterName		: STRING;
	Ptr					: POINTER TO ARRAY[0..(GPL_Component.MAX_OUTPUT_DATA_SIZE_BYTES)] OF BYTE;
	DataType			: E_DataType;
END_STRUCT
END_TYPE

// DUTs/Base/ST_PlcSystem
TYPE ST_PlcSystem EXTENDS PlcTaskSystemInfo :
STRUCT
	TaskUtilizationPercentage	: LREAL;
	LogCycleExceed				: Tc2_Standard.R_TRIG;
	LogRTViolation				: Tc2_Standard.R_TRIG;
END_STRUCT
END_TYPE

// DUTs/Command/E_CommandPriority
{attribute 'qualified_only'}
{attribute 'strict'}
{attribute 'to_string'}
TYPE E_CommandPriority :
(
    Priority_Low := 0,        // e.g., status updates
    Priority_Normal := 1,     // standard motion commands
    Priority_High := 2,       // homing, calibration
    Priority_Critical := 3    // E-Stop, safety actions
);
END_TYPE

// DUTs/Command/E_CommandResult
{attribute 'qualified_only'}
{attribute 'to_string'}
TYPE E_CommandResult :
(
	None				:= 0, //Init
	Aborted				:= 499, // new command with higher priority, etc.
	Cancelled			:= 444,  // Client cancelled before execution (custom code)
	InterlockLost		:= 424, // Command was in execute/monitor and interlock lost
    Ok                  := 200, // when de-queued
    Accepted            := 202, // when queued
 	BadRequest          := 400, // command ill-formed
    Forbidden           := 403, // lacking permissives to execute
	RequestTimeout		:= 408, 
	TooManyRequests		:= 429 // retry count exceeds what is configured for this command
) UDINT;
END_TYPE

// DUTs/Command/E_CommandState
{attribute 'qualified_only'}
{attribute 'to_string'}
TYPE E_CommandState :
(
	Idle := 0,
	Execute := 1,
	Monitor := 2,
	Paused := 3,
	Complete := 4
) UDINT;
END_TYPE

// DUTs/Command/ST_CommandConfiguration
TYPE ST_CommandConfiguration :
STRUCT
	BaseConfiguration				: REFERENCE TO ST_BaseConfiguration;
	PermIntlkConfiguration			: REFERENCE TO ST_PermIntlkConfiguration;
	CommandIndex					: DINT;
	CommandPOUName					: STRING;
	CommandDescription				: Tc2_System.T_MaxString;
	RetryCountONLYFORCOMMSENDS		: DINT := 0; // 0=no retry, 1=retry once, etc.
 	PermIntlkConfiguredAsInterlock	: BOOL := TRUE;
	AbortOnInterlockDrop			: BOOL := TRUE;
	PausedCommandRemainsBusy		: BOOL := TRUE; //No tests yet written to validate; further implementation likely required to switch configurations
	TimeoutTime						: TIME := Tc2_System.Global_Variables.DEFAULT_ADS_TIMEOUT;
	Priority						: E_CommandPriority := E_CommandPriority.Priority_Normal;
	CompletionCondition				: REFERENCE TO BOOL; // When TRUE, command transitions from Monitor to Complete state
END_STRUCT
END_TYPE

// DUTs/Command/ST_CommandStatus
TYPE ST_CommandStatus :
STRUCT
	BaseStatus						: REFERENCE TO ST_BaseStatus;
	ConfigRef						: REFERENCE TO ST_CommandConfiguration;
	LastCommandMessage				: Tc2_System.T_MaxString;
	LastCommandTriggerTime			: Tc2_Utilities.T_FILETIME64;
	LastCommandCompletionTime		: Tc2_Utilities.T_FILETIME64;
	LastCommandElapsedTime			: LTIME;
	StepState						: E_CommandState;
	CommandTryCount					: DINT;
	Result							: E_CommandResult := E_CommandResult.None;
	LastCommandResult				: E_CommandResult;
	CmdConfigurationResolution		: E_ConfigurationResolution;
	PermIntlkConfigResolution		: E_ConfigurationResolution;
	PreviousStepState				: E_CommandState; // State change detection for retry count reset
	PreviousResult					: E_CommandResult; // For preserving diagnostic info in Resume
END_STRUCT
END_TYPE

// DUTs/Component/E_ComponentTriggerMode
{attribute 'qualified_only'}
{attribute 'strict'}
{attribute 'to_string'}
TYPE E_ComponentTriggerMode :
(
	none					:= 0, //Trigger Mode Not Configured
	ExternallyTriggered 	:= 1, //Configured to be triggered by external means (not triggered by PLC)
	HardwareTriggered 		:= 2, //i.e. EtherCAT, Profinet, EIP, IO, ect.
	SoftwareTriggered 		:= 3  //i.e. ADS
) := HardwareTriggered;
END_TYPE

// DUTs/Component/ST_ComponentCommand
//TODO
//Build these into a configuration
TYPE ST_ComponentCommand :
STRUCT
	INDEX_CMD_OBTAINAMSNETID		: INT := 0;
	INDEX_CMD_ENABLE				: INT := 1;
	INDEX_CMD_DISABLE				: INT := 2;
	INDEX_CMD_RESET_ALL_CMD			: INT := 3;
	INDEX_CMD_SAVE_CONFIGURATION 	: INT := 4;
	INDEX_CMD_LOAD_CONFIGURATION 	: INT := 5;
	INDEX_CMD_RESET					: INT := 6;
	INDEX_MAX_COMPONENT_BASE		: INT := 6;
END_STRUCT
END_TYPE

// DUTs/Component/ST_ComponentConfiguration
TYPE ST_ComponentConfiguration :
STRUCT
	BaseConfiguration			: REFERENCE TO ST_BaseConfiguration;
	ResultsHandshakeEnable 		: BOOL := FALSE;
	ResultsReadyAck				: BOOL; // Used in concert with ResultsReady Handshake (must be configured TRUE)
	AmsNetIdRequired			: BOOL := TRUE;
	AmsNetId     				: Tc2_System.T_AmsNetID;
	UseCommandPriority			: BOOL := TRUE;
	ResetResetsAllCommands		: BOOL := FALSE;
END_STRUCT
END_TYPE

// DUTs/Component/ST_ComponentStatus
TYPE ST_ComponentStatus :
STRUCT
	BaseStatus						: REFERENCE TO ST_BaseStatus;
	EtherCATStatus					: ST_EtherCATStatus;	
	MethodDispatch					: DINT;
	AmsNetIdIsValid					: BOOL;	
	AmsNetId						: REFERENCE TO Tc2_System.T_AmsNetID;
	iLastCommand					: I_Command;
	iLastCommandConfiguration		: I_CommandConfiguration;
	sComponentCommandMessage		: Tc2_System.T_MaxString;
	CommandConfigurationInjected	: BOOL;
	PermIntlkConfigurationInjected	: BOOL;
END_STRUCT
END_TYPE

// DUTs/Configuration/E_ConfigurationResolution
{attribute 'qualified_only'}
{attribute 'strict'}
{attribute 'to_string'}
TYPE E_ConfigurationResolution :
(
	Local  := 0,
	InjectedInterface := 1
);
END_TYPE

// DUTs/Debounce/ST_DebounceConfiguration
TYPE ST_DebounceConfiguration :
STRUCT
	BaseConfiguration		: REFERENCE TO ST_BaseConfiguration;
	tOnDelay				: TIME;
	tOffDelay				: TIME;
//VAR_INPUT
	xRawSignal	AT %I* 		: BOOL;
	xSimSignal				: BOOL;
END_STRUCT
END_TYPE

// DUTs/Debounce/ST_DebounceStatus
TYPE ST_DebounceStatus :
STRUCT
	BaseStatus			: REFERENCE TO ST_BaseStatus;
	RefRawSignal		: REFERENCE TO BOOL;
	QRise				: BOOL;
	QFall				: BOOL;
	rtOutput			: Tc2_Standard.R_TRIG;
	ftOutput			: Tc2_Standard.F_TRIG;
//VAR_OUTPUT
	DebouncedSignal		: BOOL;
END_STRUCT
END_TYPE

// DUTs/EtherCAT/ST_EtherCATAdsAddr
//Complete ADS address to access the slave (mailbox)
TYPE ST_EtherCATAdsAddr :
STRUCT
	netId		AT %I* 	: AMSNETID;
	port		AT %I* 	: WORD;
END_STRUCT
END_TYPE

// DUTs/EtherCAT/ST_EtherCATInfoData
TYPE ST_EtherCATInfoData :
STRUCT
	State			AT %I* 	: UINT; // Same Size as Control.ST_EtherCATState Can use MEMCPY into structure
	AdsAddr			AT %I* 	: ST_EtherCATAdsAddr;
END_STRUCT
END_TYPE

// DUTs/EtherCAT/ST_EtherCATStatus
TYPE ST_EtherCATStatus :
STRUCT
	WcState			AT %I* 	: ST_EtherCATWcState; // Link to hardware
	InfoData		AT %I* 	: ST_EtherCATInfoData; // Link to hardware
	OpStatus				: ST_OpStatus;
	LinkStatus 				: E_LinkStatus;
	LinkStatusString 		: Tc2_System.T_MaxString := TO_STRING(LinkStatus);
END_STRUCT
END_TYPE

// DUTs/EtherCAT/ST_EtherCATWcState
TYPE ST_EtherCATWcState :
STRUCT
	WcState			AT %I* 	: BIT;
	InputToggle		AT %I* 	: BIT;
END_STRUCT
END_TYPE

// DUTs/EventHandling/ST_EventLogHandlerConfiguration
TYPE ST_EventLogHandlerConfiguration :
STRUCT
	BaseConfiguration	: REFERENCE TO ST_BaseConfiguration;

	// Performance Metrics Configuration
	RollingAvgWeightCurrent			: REAL := 0.1;		// Weight for current sample in rolling average (0.1 = 10%)
	RollingAvgWeightPrevious		: REAL := 0.9;		// Weight for previous average (0.9 = 90%)

	// System Health Score Weights (should sum to <= 100)
	HealthScoreUtilizationWeight	: REAL := 0.3;		// Weight for cycle utilization impact (30%)
	HealthScoreBufferWeight			: REAL := 0.4;		// Weight for buffer utilization impact (40%)
	HealthScorePersistencePenalty	: REAL := 20.0;		// Penalty when persistence failures occur
	HealthScoreCycleExceedPenalty	: REAL := 10.0;		// Penalty when cycle time exceeded

	// Exponential Backoff Configuration (milliseconds)
	BackoffInitialDelayMs			: UDINT := 100;		// Initial backoff delay
	BackoffMaxDelayMs				: UDINT := 10000;	// Maximum backoff delay (10 seconds)
	BackoffMultiplier				: REAL := 2.0;		// Backoff multiplier for exponential growth
	MaxRetryAttemptsPerEntry		: UINT := 5;		// Maximum retry attempts for a single entry before discarding

	// Dynamic Rate Control - Task Utilization Thresholds
	TaskUtilHighThreshold			: REAL := 0.8;		// High load threshold (80% - uses LOG_CYCLE_EXCEED_MAX_THRESHOLD)
	TaskUtilModerateThreshold		: REAL := 0.6;		// Moderate load threshold (60%)
	TaskUtilLowThreshold			: REAL := 0.3;		// Low load threshold (30%)

	// Dynamic Rate Control - Rate Divisors/Multipliers
	RateDivisorHighLoad				: UDINT := 4;		// Divide rate by 4 under high load
	RateDivisorModerateLoad		: UDINT := 2;		// Divide rate by 2 under moderate load
	RateMultiplierLowLoad			: UDINT := 2;		// Multiply rate by 2 under low load

	// Dynamic Rate Control - Buffer Thresholds
	BufferThresholdEmergency		: REAL := 95.0;		// Emergency mode threshold (95%)
	BufferThresholdHigh				: REAL := 90.0;		// High buffer threshold (90%)
	BufferThresholdIncrease			: REAL := 80.0;		// Threshold to increase rate under low load (80%)

	// Dynamic Rate Control - Emergency Multipliers
	EmergencyRateMultiplier			: UDINT := 3;		// Rate multiplier for emergency mode
	HighBufferRateMultiplier		: UDINT := 2;		// Rate multiplier for high buffer usage

	// Dynamic Rate Control - Absolute Limits
	MaxEntriesPerScanAbsolute		: UINT := 200;		// Absolute maximum entries per scan
END_STRUCT
END_TYPE

// DUTs/EventHandling/ST_EventLogHandlerStatus
TYPE ST_EventLogHandlerStatus :
STRUCT
	BaseStatus		: REFERENCE TO ST_BaseStatus;
	// Core operational variables
	LogCountThisScan		: UINT;					// Entries processed this scan cycle
	ShouldProcess			: BOOL;					// Determines if dequeue should run
	DynamicMaxEntries		: UINT;					// Calculated max entries per scan
	PersistenceSuccess		: BOOL;					// Result of AddToEventLog call
	CycleStartTime			: UDINT;				// Start time for performance metrics
	ExitProcessing			: BOOL;
	CurrentEntryRetryCount	: UINT;					// Number of retries for current entry being processed

	// Consolidated state structures
	LoggingMetrics			: ST_LogMetrics;		// Comprehensive logging metrics
	BackoffState			: ST_LogBackoffState;	// Persistence failure backoff state

	// Edge detection
	BufferOverflowTrigger	: R_TRIG;				// Edge detection for buffer overflow

	// Cycle break protection
	ConsecutiveRemoveFailures	: UINT;				// Count of consecutive RemoveObject failures
	ConsecutiveEmptyScans		: UINT;				// Scans with no successful processing
	LastSuccessfulProcessTime	: UDINT;			// Timestamp of last successful entry processing
	BufferCorruptionDetected	: BOOL;				// Flag indicating buffer state corruption
	ForceBufferReset			: BOOL;				// Trigger to force reset corrupted buffer
END_STRUCT
END_TYPE

// DUTs/EventHandling/ST_PersistentStorageStatus
TYPE ST_PersistentStorageStatus :
STRUCT
	BaseStatus					: REFERENCE TO ST_BaseStatus;
	MessagesSentThisScan		: UDINT;
	Previous_AddEntrySource		: T_MaxString;
	Previous_AddEntryMessage	: T_MaxString;
	Previous_AddEntryFlags		: UDINT;
	NotInitializedMessageShown	: BOOL;

	// Duplicate suppression tracking
	DuplicateSuppressionCount	: UINT;		// Number of consecutive duplicates suppressed
	LastUniqueMessageTime		: ULINT;	// Timestamp when last unique message was sent (FILETIME format)
	ConsecutiveDuplicateLimit	: UINT := 10;	// Max duplicates to suppress before allowing through
END_STRUCT
END_TYPE

// DUTs/File/Structs/ST_AmsNetId
TYPE ST_AmsNetId :
STRUCT
	AmsNetIdIsValid			: BOOL;
	AmsNetIdStr				: Tc2_System.T_AmsNetID;
	AmsNetIdBytes			: Tc2_System.T_AmsNetIdArr;
	GetAmsNetIdBusy			: BOOL;
	GetAmsNetIdError		: BOOL;
	GetAmsNetIdErrorId		: UDINT;  
END_STRUCT
END_TYPE

// DUTs/File/Structs/ST_FileHandlerBaseStatus
TYPE ST_FileHandlerBaseStatus :
STRUCT
	ComponentStatus			: REFERENCE TO ST_ComponentStatus;
//	FileOpStatus            : ARRAY[GPL_File.MIN_INDEX_FILEOP..GPL_File.MAX_INDEX_FILEOP] OF ST_FileOpStat;
END_STRUCT
END_TYPE

// DUTs/File/Structs/ST_FileHandlerConfiguration
TYPE ST_FileHandlerConfiguration :
STRUCT
	ComponentConfiguration			: REFERENCE TO ST_ComponentConfiguration;
	FileFormat						: E_FileFormat				:= E_FileFormat.CSV;
	Enable							: BOOL 						:= TRUE;
	LoggerUpdateMinInterval			: TIME 						:= T#20MS;
	LoggerUpdateMaxInterval			: TIME 						:= T#500MS;	
	FileLogName						: Tc2_System.T_MaxString  	:= GPL_File.FileLogPath;
	NewLineChar						: STRING(4) 				:= GPL_File.NewLineChar;
	Delimiter						: STRING(2)					:= GPL_File.Delimiter;
	LineNumberChar					: STRING(4) 				:= 'LN';
	Timestamp						: STRING(10)				:= 'Timestamp';
	MaxFileNumber					: UINT      				:= 3;
	Timeout							: TIME      				:= Tc2_System.DEFAULT_ADS_TIMEOUT;
	FileNameSuffix					: Tc2_System.T_MaxString	:= GPL_File.FileExtension;
	BeckhoffFileOpPath				: Tc2_System.E_OpenPath 	:= GPL_File.BeckhoffFileOpPath;
	BeckhoffFileOpMode				: DWORD						:= Tc2_System.Global_Variables.FOPEN_MODEAPPEND;
END_STRUCT
END_TYPE

// DUTs/File/Structs/ST_FileHandlerCSVConfiguration
TYPE ST_FileHandlerCSVConfiguration :
STRUCT
	BaseFileHandleConfiguration		: REFERENCE TO ST_FileHandlerConfiguration;
	FileFormat						: E_FileFormat				:= E_FileFormat.CSV;
	Enable							: BOOL 						:= TRUE;
	LoggerUpdateMinInterval			: TIME 						:= T#20MS;
	LoggerUpdateMaxInterval			: TIME 						:= T#500MS;	
	FileLogName						: Tc2_System.T_MaxString  	:= GPL_File.FileLogPath;
	NewLineChar						: STRING(4) 				:= GPL_File.NewLineChar;
	Delimiter						: STRING(2)					:= GPL_File.Delimiter;
	LineNumberChar					: STRING(4) 				:= 'LN';
	Timestamp						: STRING(10)				:= 'Timestamp';
	MaxFileNumber					: UINT      				:= 3;
	Timeout							: TIME      				:= Tc2_System.DEFAULT_ADS_TIMEOUT;
	FileNameSuffix					: Tc2_System.T_MaxString	:= GPL_File.FileExtension;
	BeckhoffFileOpPath				: Tc2_System.E_OpenPath 	:= GPL_File.BeckhoffFileOpPath;
	BeckhoffFileOpMode				: DWORD						:= Tc2_System.Global_Variables.FOPEN_MODEAPPEND;
END_STRUCT
END_TYPE

// DUTs/File/Structs/ST_FileHandlerCSVStatus
TYPE ST_FileHandlerCSVStatus :
STRUCT
	FileHandlerStatus		: REFERENCE TO ST_FileHandlerBaseStatus;
	FileHandle				: UINT;
	FileIsOpen				: BOOL;
	cbWritten				: UDINT;
	nElementsToWrite		: UDINT;
END_STRUCT
END_TYPE

// DUTs/File/Structs/ST_FileHandlerJsonStatus
TYPE ST_FileHandlerJsonStatus :
STRUCT
	FileHandlerStatus              : REFERENCE TO ST_FileHandlerBaseStatus;
	//json specific stuff
	JsonRef					: Global.SJsonValue;
END_STRUCT
END_TYPE

// DUTs/File/Structs/ST_FileOpStatus
TYPE ST_FileOpStatus :
STRUCT
//	Done					: BOOL;
	Timeout					: Tc2_Standard.TON := (PT := Tc2_System.DEFAULT_ADS_TIMEOUT);
	rtDone					: Tc2_Standard.R_TRIG;
	ftBusy					: Tc2_Standard.F_TRIG;
// 	StartTimeStamp			: ULINT;
// 	EndTimestamp			: ULINT;
// 	OpElapsedTime      		: ULINT;
	ActiveFileHandleID		: ULINT; //could be SJsonValue or UDINT returned by Beckhoff FileOp Function Blocks, for example
	pBuffer					: Global.PVOID;
	FileOpByteCount			: UDINT;
	FileOpPath				: Tc2_System.T_MaxString;
END_STRUCT
END_TYPE

// DUTs/File/E_FileFormat
{attribute 'qualified_only' := ''}
{attribute 'strict' := ''}
{attribute 'to_string' := ''}
TYPE E_FileFormat :
(
	CSV   := 0,
	JSON  := 1,
 	XML   := 2
) USINT;
END_TYPE

// DUTs/Hash/ST_HashTableConfiguration
TYPE ST_HashTableConfiguration :
STRUCT
	BaseConfiguration	: REFERENCE TO ST_BaseConfiguration;
	Capacity     		: UINT := GPL_HashTable.INDEX_MAX - GPL_HashTable.INDEX_MIN +1;             // must be power‐of‐two
	LoadFactor      	: REAL := 0.75;             // guard threshold
END_STRUCT
END_TYPE

// DUTs/Hash/ST_HashTableStatus
TYPE ST_HashTableStatus :
STRUCT
	BaseStatus		: REFERENCE TO ST_BaseStatus;
	Count			: UINT;        			// number of live entries
	Capacity		: REFERENCE TO UINT;         // current bucket count
	LoadFactor		: REFERENCE TO REAL;         // Count / Capacity
	HashTableIsPowerOf2	: BOOL;
END_STRUCT
END_TYPE

// DUTs/LogTrace/E_LogTraceWhen
{attribute 'qualified_only'}
{attribute 'strict'}
{attribute 'to_string'}
TYPE E_LogTraceWhen :
(
	xRunOnInitOnly := 0,
	xRunCyclic := 1
);
END_TYPE

// DUTs/LogTrace/ST_LogBackoffState
TYPE ST_LogBackoffState :
STRUCT
	PersistenceFailureCount		: UINT;				// Number of consecutive persistence failures
	BackoffTimer				: TON;				// Timer for exponential backoff
	BackoffDelayMs				: UDINT;			// Current backoff delay in milliseconds
	PersistenceBlocked			: BOOL;				// TRUE when in backoff state
END_STRUCT
END_TYPE

// DUTs/LogTrace/ST_LogMetrics
TYPE ST_LogMetrics :
STRUCT
	// Performance metrics
	CycleUtilizationPercentage			: LREAL;					// Current cycle utilization (0-100%)
	AverageProcessingTimeMs				: REAL;					// Average processing time per cycle
	PeakProcessingTimeMs				: UDINT;				// Peak processing time observed

	// Throughput metrics
	EntriesProcessedThisCycle			: UINT;					// Entries processed in current cycle
	EntriesProcessedPerSecond			: REAL;					// Rolling average entries/sec
	TotalEntriesProcessed				: UDINT;				// Total entries processed since boot

	// Buffer health metrics
	BufferUtilizationPercentage			: REAL;					// Buffer fill level (0-100%)
	MaxBufferUtilizationReached			: REAL;					// Peak buffer utilization seen
	BufferOverflowCount					: UDINT;				// Number of buffer overflows

	// Failure and backoff metrics
	PersistenceFailureCount				: UDINT;				// Total persistence failures
	BackoffActiveCount					: UDINT;				// Times backoff was activated
	CurrentBackoffDelayMs				: UDINT;				// Current backoff delay
	TotalBackoffTimeMs					: UDINT;				// Total time spent in backoff

	// Severity distribution metrics
	CriticalEntriesProcessed			: UDINT;				// Count of critical entries
	ErrorEntriesProcessed				: UDINT;				// Count of error entries
	WarningEntriesProcessed				: UDINT;				// Count of warning entries
	InfoEntriesProcessed				: UDINT;				// Count of info entries

	// System health indicators
	CycleExceedCount					: UDINT;				// Number of cycle exceeds in logging task
	SystemHealthScore					: REAL;					// Overall system health (0-100%)
	LastResetTimestamp					: UDINT;				// When metrics were last reset
END_STRUCT
END_TYPE

// DUTs/LogTrace/ST_LogTraceConfiguration
TYPE ST_LogTraceConfiguration :
STRUCT
	What	: ST_LogTraceWhat;
	When	: E_LogTraceWhen := E_LogTraceWhen.xRunOnInitOnly;
END_STRUCT
END_TYPE

// DUTs/LogTrace/ST_LogTraceStatus
TYPE ST_LogTraceStatus :
STRUCT
	MessageShown						: BOOL;
	InitChildrenFailureShown			: BOOL;
	InitReferencesFailureShown			: BOOL;
	InitDependencyConfigFailureShown	: BOOL;
	CmdConfigStashedShown           	: BOOL;
	PermIntlkConfigStashedShown     	: BOOL;
	PermIntlkConfigInjectedShown    	: BOOL;
	CmdConfigInjectedShown          	: BOOL;
	PermIntlkInitializedShown       	: BOOL;
	DependencyConfigSetShown        	: BOOL;
	ConfigsInjectedToChildrenShown  	: BOOL;
	ComponentInterfaceInjectedShown 	: BOOL;
	CmdConfigInterfaceInjectedShown 	: BOOL;
	CmdConfigToPermIntlkShown       	: BOOL;
	ChildDepsInitializedShown       	: BOOL;
	// Cyclic validation and monitoring message flags
	CmdValidatedShown               	: BOOL;	// Suppress "Idle/Executing/Paused/Completed command validated"
	CmdValidationFailedShown        	: BOOL;	// Suppress "Command validation failed: Forbidden"
	CompletionConditionMetShown     	: BOOL;	// Suppress "Completion condition met"
	InterlockLossShown              	: BOOL;	// Suppress interlock loss messages during monitoring
	PermIntlkConditionFailureShown  	: BOOL;	// Suppress permissive condition failure messages
	ConfigInvalidRefShown           	: BOOL;	// Suppress configuration invalid reference messages
END_STRUCT
END_TYPE

// DUTs/LogTrace/ST_LogTraceWhat
TYPE ST_LogTraceWhat :
STRUCT
	xLogToAdsConsole 	: BOOL := FALSE;
	xLogToEventLogger 	: BOOL := TRUE;
	xLogToFile 			: BOOL := FALSE;
	MinTraceLevel		: Global.TcEventSeverity := Global.TcEventSeverity.Warning;
END_STRUCT
END_TYPE

// DUTs/PermIntlk/E_ModePermIntlk
{attribute 'qualified_only'}
{attribute 'strict'}
TYPE E_ModePermIntlk :
(
	IfAllConditionsMet  := 0,
	IfAnyConditionMet   := 1
) := IfAllConditionsMet;
END_TYPE

// DUTs/PermIntlk/ST_PermIntlkConfiguration
TYPE ST_PermIntlkConfiguration :
STRUCT
	BaseConfiguration		: REFERENCE TO ST_BaseConfiguration;
	Mode          			: E_ModePermIntlk;
	PermIntlkObj			: ARRAY[GC_PermIntlk.INDEX_CONDITION_MIN..GC_PermIntlk.INDEX_CONDITION_MAX] OF ST_PermIntlkConfigurationCondition; 
END_STRUCT
END_TYPE

// DUTs/PermIntlk/ST_PermIntlkConfigurationCondition
TYPE ST_PermIntlkConfigurationCondition :
STRUCT
	Index		: DINT;
	Description : STRING(GPL_PermIntlk.DESCRIPTION_LEN) := 'PermIntlk Condition Not Configured'; //Functional description of the condition
	Condition  	: REFERENCE TO BOOL; //A condition that must evaluate to true for this permintlk to be OK. TRUE by default in the case it was not set.
//	Bypassable	: BOOL := FALSE; //Is this permintlk bypassable?
END_STRUCT
END_TYPE

// DUTs/PermIntlk/ST_PermIntlkStatus
TYPE ST_PermIntlkStatus :
STRUCT
	BaseStatus						: REFERENCE TO ST_BaseStatus;
	ConfigRef						: REFERENCE TO ARRAY[GC_PermIntlk.INDEX_CONDITION_MIN..GC_PermIntlk.INDEX_CONDITION_MAX] OF ST_PermIntlkConfigurationCondition;
	PermissiveStatusMessage 		: Tc2_System.T_MaxString;
	ConditionStatus					: ARRAY[GC_PermIntlk.INDEX_CONDITION_MIN..GC_PermIntlk.INDEX_CONDITION_MAX] OF ST_PermIntlkStatusCondition;
	PermIntlkOK   					: BOOL := TRUE;
	PermIntlkConfigResolution		: E_ConfigurationResolution;
	PermIntlkConditionAlwaysFalse	: BOOL; // do not initialize TRUE
END_STRUCT
END_TYPE

// DUTs/PermIntlk/ST_PermIntlkStatusCondition
TYPE ST_PermIntlkStatusCondition :
STRUCT
	PermObj				: REFERENCE TO ST_PermIntlkConfigurationCondition;
	Configured			: BOOL := FALSE; //Is Index configured
	ConditionMessage 	: Tc2_System.T_MaxString;
END_STRUCT
END_TYPE

// DUTs/RingBuffer/ST_LogEntry
TYPE ST_LogEntry :
STRUCT
	systimestamp	: ULINT;
	Message			: Tc2_System.T_MaxString;
	Severity		: Global.TcEventSeverity;
	RaiseAlarm		: BOOL := FALSE;
	InstancePath	: STRING;
	TaskInfo		: PlcTaskSystemInfo;
	RetryCount		: UINT := 0;				// Number of times persistence has been retried for this entry
END_STRUCT
END_TYPE

// DUTs/RingBuffer/ST_RingBufferCfg
TYPE ST_RingBufferCfg :
STRUCT
	BaseConfiguration		: REFERENCE TO ST_BaseConfiguration;
	CopyToLargeMemoryArea   : BOOL := TRUE;
	CopyOnlyUniqueMessage   : BOOL := FALSE;
	AllowOverwriteSecBuffer : BOOL := FALSE;
	ByteCountOfDataObj      : UDINT; // do not write to this manually; done using SIZEOF function
	WriteDataToFile         : BOOL := FALSE;
	RemoveAfterAdd			: BOOL;
	ReadByteOffset			: UDINT;
END_STRUCT
END_TYPE

// DUTs/RingBuffer/ST_RingBufferStatus
TYPE ST_RingBufferStatus :
STRUCT
	BaseStatus					: REFERENCE TO ST_BaseStatus;
	GlobalCounter				: UDINT;
	ObjectCountInBufferPrim		: UDINT;
	BufferIsFullPrim        	: BOOL;
	ObjectWasAddedPrimary   	: BOOL;
	ObjectWasRemovedPrimary 	: BOOL;
	ObjectWasPeekedPrimary		: BOOL;
	ObjectWasReadPrimary		: BOOL;
	Overwriting             	: BOOL;
	ByteCountInBufferPrim   	: ULINT;  
	BufferCapacity          	: UDINT;
	CountBytesWritten			: ULINT;
	CountBytesRemoved			: UDINT;
	CountBytesCleared			: UDINT;
	CountBytesPeeked			: UDINT;
	CountBytesRead				: UDINT;
	WillOverwrite    			: BOOL;
END_STRUCT
END_TYPE

// DUTs/RingBuffer/ST_SystimeICmd
TYPE ST_SystimeICmd :
STRUCT
  systimestamp		: ULINT;    // system timestamp
  iCmd				: I_Command;
  iCmdCfg			: I_CommandConfiguration;
END_STRUCT
END_TYPE

// DUTs/RingBuffer/ST_SystimeString
TYPE ST_SystimeString :
STRUCT
  systimestamp   : ULINT;    // system timestamp
  stringval      : STRING(GPL_RingBuffer.STRING_LENGTH);
END_STRUCT
END_TYPE

// DUTs/Safety/ST_SafetyGroupConfiguration
TYPE ST_SafetyGroupConfiguration :
STRUCT
	BaseConfiguration 			: REFERENCE TO ST_BaseConfiguration;
	RunStop			AT %Q*		: BOOL	:= TRUE;
	ErrAck			AT %Q*		: BOOL;
//	ModuleFault		AT %Q*		: BOOL;
END_STRUCT
END_TYPE

// DUTs/Safety/ST_SafetyGroupStatus
TYPE ST_SafetyGroupStatus :
STRUCT
	BaseStatus					: REFERENCE TO ST_BaseStatus;
	FBErr				AT %I*	: BOOL;
	ComErr				AT %I*	: BOOL;
//	OutErr				AT %I*	: BOOL;
	OtherErr			AT %I*	: BOOL;
// 	ComStartup			AT %I*	: BOOL;
// 	FBDeactive			AT %I*	: BOOL;
	FBRun				AT %I*	: BOOL;
	InRun				AT %I*	: BOOL;
	SafetyGroupOK		AT %I*	: BOOL;
	State				AT %I* 	: BOOL;
	Diag				AT %I* 	: BOOL;
END_STRUCT
END_TYPE

// DUTs/Sequencer/E_Operation
{attribute 'strict'}
{attribute 'to_string'}
{attribute 'qualified_only'}
TYPE E_Operation :
(
    NOP := 0,

    // --- Top Chuck Z Moves (10–19) ---
    TopChuck_DownToFoil := 10,           // down to foil position
    TopChuck_DownToWafer := 11,          // down to wafer position
    TopChuck_RapidHome := 12,             // up to Z home
    TopChuck_MethodicalSlowCarefulLiftup := 13,         // param[1]=distance (mm, e.g. 3), fixed velocity = 1 mm/s

    // --- Top Chuck Lateral Moves (20–29) ---
    TopChuck_Lateral_Home := 20,         // lateral home station
    TopChuck_Lateral_Laser := 21,         // lateral position over foil station
    TopChuck_Lateral_Wafer := 22,        // lateral position over wafer station

    // --- Top Chuck Utilities (30–39) ---
    TopChuck_VacuumOn := 30,
    TopChuck_VacuumOff := 31,
    TopChuck_PurgeOn := 32,
    TopChuck_PurgeOff := 33,
    TopChuck_ElectrostaticOn := 34,      // param[1]=voltage (V), param[2]=mode (0=monopolar, 1=bipolar)
    TopChuck_ElectrostaticOff := 35,

    // --- Bottom Chuck Operations (40–49) ---
	
    BottomChuck_Up := 40,             // param[1]=position (mm)
    BottomChuck_Down := 41,             // param[1]=position (mm)
    BottomChuck_ElectrostaticOn := 42,   // param[1]=voltage (V), param[2]=mode (0=mono,1=bi)
    BottomChuck_ElectrostaticOff := 43,

    // --- Web / Foil Handling (50–59) ---
    WebDrive_ApplyTension := 50,           // param[1]=tension (N) (tensies)
    WebDrive_ScrollFoil := 51,           // param[1]=distance (mm) or speed (mm/s)

    // --- Microscope / Zaber Axes (60–69) ---
    WaferChuckX_Move := 60,                   // param[1]=position (mm), param[2]=velocity (mm/s)
    WaferChuckY_Move := 61,                   // param[1]=position (mm), param[2]=velocity (mm/s)
    WaferChuckTheta_Move := 62,               // param[1]=angle (deg), param[2]=velocity (deg/s)

    // --- Vision / Scanning (70–79) ---
    Vision_Run := 70,                    // param[1]=routineID, param[2]=timeout (s)

    // --- Laser Cutting Placeholders (80–89) ---
    Laser_VerticalCut := 80,             // placeholder, executed outside PLC
    Laser_EndCut := 81,                  // placeholder, executed outside PLC

    // --- Utility (100–109) ---
    Wait := 100                          // Timeout field in ST_Operation used directly

    // =====================================================================
    // Operator-only steps (not automated, for documentation only)
    // =====================================================================
    // Soldering (Operator)
    // Doors_Open (Operator)
    // Doors_Close (Operator)
    // Place strate (Operator)
    // Place Wafer (Operator)
    // WaferVacuum (Operator)
    // Place paper (Operator)
    // Align foil manually (Operator)
    // Calibration chuck (Operator) – bipolar +2000/-2000
    // Smoothing (Operator)
    // Cleaning strate AlN with IPA (Operator)
    // Cleaning strate AlN with air gun (Operator)
    // Placing Cu block weight on cuts by hand (Operator)
    // Remove weight (Operator)
    // Place Gorilla Glass (Operator)
    // Turn off bottom chuck vacuum (Operator)
);
END_TYPE

// DUTs/Sequencer/E_PackMLState
{attribute 'qualified_only'}
{attribute 'to_string'}
TYPE E_PackMLState :
(
	Idle			:= 0, // Machine is powered AND initialized, but NOT producing.
	Starting		:= 1, // Transition FROM Idle TO Execute (preparing FOR operation).
	Execute			:= 2, // Actively running / producing.
	Completing		:= 3, // Finalizing current cycle OR lot before stopping.
	Complete		:= 4, // Finished with work, no further execution.
	Stopping		:= 5, // Controlled stop in progress.
	Stopped			:= 6, // Machine stopped (NOT running).
	Aborting		:= 7, // Emergency stop OR uncontrolled shutdown.
	Aborted			:= 8, // Machine halted due TO fault OR error.
	Clearing		:= 9, // Transition TO clear aborts/faults, prepare TO reset.
	Resetting		:= 10, // Transition TO Idle (re-initialize).
	Holding			:= 11, // Initiating pause in execution.
	Held			:= 12, // Execution paused, ready TO resume.
	Unholding		:= 13, // Transition FROM Held back TO Execute.
	Suspending		:= 14, // Initiating suspension (often external condition, e.g., upstream starved).
	Suspended		:= 15, // Execution suspended, waiting FOR condition TO clear.
	Unsuspending	:= 16 // Transition FROM Suspended back TO Execute.
);
END_TYPE

// DUTs/Sequencer/ST_Operation
TYPE ST_Operation :
	STRUCT
		HMILabel	 : STRING; 			//'Move Gantry Stage to Home Position'
		OperationID  : E_Operation;  	// enum: MoveAxis, VisionCheck, HVTest, LoadWafer, etc.
		AxisID       : INT;              // if motion: which axis
		Position     : LREAL;            // target position
		Velocity     : LREAL;            // optional
		Timeout      : TIME;             // max duration allowed
		Parameters   : ARRAY[GPL_Recipe.INDEX_OPPARAM_MIN..GPL_Recipe.INDEX_OPPARAM_MAX] OF LREAL; // generic parameter (voltage, threshold) - define in spreadsheet/csv
	END_STRUCT
END_TYPE

// DUTs/Sequencer/ST_OperationSequencerConfiguration
TYPE ST_OperationSequencerConfiguration :
STRUCT
	ComponentConfiguration				: REFERENCE TO ST_ComponentConfiguration;
END_STRUCT
END_TYPE

// DUTs/Sequencer/ST_OperationSequencerStatus
TYPE ST_OperationSequencerStatus :
STRUCT
	ComponentStatus				: REFERENCE TO ST_ComponentStatus;	
	CurrentState				: E_PackMLState;
	NewState					: E_PackMLState;
	CommandResult				: E_CommandResult;
    // Step execution state
    StepTimeout             : TON;          // timeout timer for current step
    StepStarted             : BOOL := FALSE;
    StepDone                : BOOL := FALSE;
    StepError               : BOOL := FALSE;
    SequenceComplete        : BOOL := FALSE;

    // Diagnostics
    ErrorCode               : DINT := 0;
    FaultOpID               : E_Operation := E_Operation.NOP;
END_STRUCT
END_TYPE

// DUTs/Sequencer/ST_PackMLSequencerConfiguration
TYPE ST_PackMLSequencerConfiguration :
STRUCT
	ComponentConfiguration				: REFERENCE TO ST_ComponentConfiguration;
END_STRUCT
END_TYPE

// DUTs/Sequencer/ST_PackMLSequencerStatus
TYPE ST_PackMLSequencerStatus :
STRUCT
	ComponentStatus				: REFERENCE TO ST_ComponentStatus;
	CurrentState				: E_PackMLState;
	NewState					: E_PackMLState;
	PreviousState				: E_PackMLState;	// Track state from previous cycle for auto-transitions
	CommandResult				: E_CommandResult;
END_STRUCT
END_TYPE

// Base/GC_Base
{attribute 'qualified_only'}
{attribute 'global_init_slot' := '40600'}
VAR_GLOBAL CONSTANT
	CountOf100NsIncrement1Hr  		: LINT  := 36000000000;  // do not edit
	// Unit Conversion Constants
	MillisecondsPerSecond			: REAL := 1000.0;	// For ms to seconds conversion
	PercentageMultiplier			: REAL := 100.0;	// For decimal to percentage conversion
END_VAR

// Base/GPL_Base
{attribute 'qualified_only'}
{attribute 'global_init_slot' := '40500'}
VAR_GLOBAL CONSTANT
	xLogToAdsConsole					: BOOL := FALSE;
	xLogToEventLogger					: BOOL := TRUE;
	xLogToFile							: BOOL := FALSE;
	eLogWhen							: E_LogTraceWhen := E_LogTraceWhen.xRunOnInitOnly;
	HourDeltaFromUtc					: SINT  := -7;
	ClockIntervalPlcSystem				: UDINT := 2;
	TRACING_ENABLED						: BOOL	:= TRUE;
	MAX_LOG_ENTRIES_PER_SCAN			: UDINT := 50;
	LOG_CYCLE_EXCEED_MAX_THRESHOLD		: LREAL := 0.7;
	PERSISTENT_LOG_LEVEL_MIN			: Global.TcEventSeverity := Global.TcEventSeverity.Warning;
	ALLOW_DUPLICATE_SEQUENTIAL_MESSAGES : BOOL	:= FALSE;
	INDEX_MIN_TASK						: DINT := 0;
	INDEX_MOTION_TASK					: DINT := 0;
	INDEX_PLC_TASK						: DINT := 1;
	INDEX_TEST_TASK						: DINT := 2;
	INDEX_LOG_TASK						: DINT := 3;
	INDEX_MAX_TASK						: DINT := 3;
END_VAR

// Component/GVLs/GC_Component
{attribute 'qualified_only'}
{attribute 'global_init_slot' := '40601'}
VAR_GLOBAL CONSTANT
	INDEX_COMMAND_MIN		: DINT := GPL_Component.INDEX_COMMAND_MIN;
	INDEX_COMMAND_MAX		: DINT := GPL_Component.INDEX_COMMAND_MAX;
END_VAR

// Component/GVLs/GPL_Component
{attribute 'qualified_only'}
{attribute 'global_init_slot' := '40501'}
VAR_GLOBAL CONSTANT
	MAX_OUTPUT_DATA_SIZE_BYTES		: DINT := 1023;
	INDEX_COMMAND_MIN				: DINT := 0;
	INDEX_COMMAND_MAX				: DINT := 3;
END_VAR

// ControlMode/GVLs/GC_ControlMode
{attribute 'qualified_only'}
{attribute 'global_init_slot' := '40602'}
VAR_GLOBAL CONSTANT
	INDEX_COMMAND_MIN		: DINT := GPL_ControlMode.INDEX_COMMAND_MIN;
	INDEX_COMMAND_MAX		: DINT := GPL_ControlMode.INDEX_COMMAND_MAX;	
END_VAR

// ControlMode/GVLs/GPL_ControlMode
{attribute 'qualified_only'}
{attribute 'global_init_slot' := '40502'}
VAR_GLOBAL CONSTANT
	INDEX_COMMAND_MIN		: DINT := 0;	
	INDEX_COMMAND_MAX		: DINT := 1;
END_VAR

// EventHandling/GVL_System
{attribute 'qualified_only'}
{attribute 'global_init_slot' := '40100'}
VAR_GLOBAL
	GlobalEventLog		: FB_PersistentEventLog;
	iPersistentStorage	: I_PersistentStorage := GlobalEventLog;

	RingBufferLog		: FB_RingBufferLogEntry;
	iBuffer				: I_RingBufferLogEntry := RingBufferLog;

	EventLogHandler		: FB_EventLogHandler;
	PlcSystemInfo 		: ARRAY[GPL_Base.INDEX_MIN_TASK..GPL_Base.INDEX_MAX_TASK] OF ST_PlcSystem;

	// Re-entry guard to prevent infinite recursion in logging subsystem
	InReentry_Logging	: BOOL := FALSE;
END_VAR

// File/GC_File
{attribute 'qualified_only'}
{attribute 'global_init_slot' := '40607'}
VAR_GLOBAL CONSTANT
	INDEX_COMMAND_MIN	: DINT := GPL_File.INDEX_COMMAND_MIN;
	INDEX_COMMAND_MAX	: DINT := GPL_File.INDEX_COMMAND_MAX;
	
	INDEX_OPENFILE		: DINT := GPL_File.INDEX_OPENFILE;
	INDEX_CLOSEFILE		: DINT := GPL_File.INDEX_CLOSEFILE;
	INDEX_READFILE		: DINT := GPL_File.INDEX_READFILE;
	INDEX_WRITEFILE		: DINT := GPL_File.INDEX_WRITEFILE;
	INDEX_RENAMEFILE	: DINT := GPL_File.INDEX_RENAMEFILE;
	INDEX_APPENDTOFILE	: DINT := GPL_File.INDEX_APPENDTOFILE;
	INDEX_CREATEFILE	: DINT := GPL_File.INDEX_CREATEFILE;
	INDEX_DELETEFILE	: DINT := GPL_File.INDEX_DELETEFILE;
END_VAR

// File/GPL_File
{attribute 'qualified_only'}
{attribute 'global_init_slot' := '40507'}
VAR_GLOBAL CONSTANT
	INDEX_COMMAND_MIN			: DINT := 0;
	INDEX_COMMAND_MAX			: DINT := 9;

	/// The log file path under 
	FileLogPath					: Tc2_System.T_MaxString := 'C:\LogFiles\Log_';
	/// Maximum string length for entering log message. Upper limit is 1500 characters
	MAX_LOG_ENTRY_STRING_LEN	: UINT := 255;

	BeckhoffFileOpPath        	: Tc2_System.E_OpenPath := E_OpenPath.PATH_GENERIC;
	BeckhoffFileOpMode			: DWORD; // := Tc2_System.Global_Variables.FOPEN_MODEAPPEND;

	udiMaxFileLogLines  		: UDINT	:= 100000;	(* Defines the max number of lines in each log file *)
	
	Delimiter					: STRING(2)		:= ',';
	FileExtension				: STRING(10)	:= '.csv';
	NewLineChar					: STRING(4)		:= '$N';
	
	INDEX_OPENFILE				: DINT := 0;
	INDEX_CLOSEFILE				: DINT := 1;
	INDEX_READFILE				: DINT := 2;
	INDEX_WRITEFILE				: DINT := 3;
	INDEX_RENAMEFILE			: DINT := 4;
	INDEX_APPENDTOFILE			: DINT := 5;
	INDEX_CREATEFILE			: DINT := 6;
	INDEX_DELETEFILE			: DINT := 7;
END_VAR

// Hashing/GPL_HashTable
{attribute 'qualified_only'}
VAR_GLOBAL CONSTANT
	INDEX_MIN	: UINT := 0;
	INDEX_MAX	: UINT := 1023; // make a power of 2 with a 0 MIN (IE. MAX-MIN = 2^X)
END_VAR

// PermIntlk/GVLs/GC_PermIntlk
{attribute 'qualified_only'}
{attribute 'global_init_slot' := '40606'}
VAR_GLOBAL CONSTANT
	INDEX_CONDITION_MIN		: DINT := GPL_PermIntlk.INDEX_CONDITION_MIN;
	INDEX_CONDITION_MAX		: DINT := GPL_PermIntlk.INDEX_CONDITION_MAX;
END_VAR

// PermIntlk/GVLs/GPL_PermIntlk
{attribute 'qualified_only'}
{attribute 'global_init_slot' := '40506'}
VAR_GLOBAL CONSTANT
	INDEX_CONDITION_MIN 	: UINT := 0;	
	INDEX_CONDITION_MAX 	: UINT := 4;
	DESCRIPTION_LEN 		: UINT := 255;
END_VAR

// RingBuffer/GVLs/GPL_RingBuffer
{attribute 'qualified_only'}
VAR_GLOBAL CONSTANT
	MIN_NUMBER_OBJECTS 	: UDINT := 0;
	MAX_NUMBER_OBJECTS 	: UDINT := 4;
	STRING_LENGTH		: UINT := 49;
	MIN_LOGENTRIES 		: UDINT := 0;
	MAX_LOGENTRIES 		: UDINT := 5999;
END_VAR

// Safety/GVLs/GC_Safety
{attribute 'qualified_only'}
{attribute 'global_init_slot' := '40605'}
VAR_GLOBAL CONSTANT
	INDEX_DEVICE_MIN 	: UINT := GPL_Safety.INDEX_DEVICE_MIN;	
	INDEX_DEVICE_MAX 	: UINT := GPL_Safety.INDEX_DEVICE_MAX;
	INDEX_GROUP_MIN 	: UINT := GPL_Safety.INDEX_GROUP_MIN;	
	INDEX_GROUP_MAX 	: UINT := GPL_Safety.INDEX_GROUP_MAX;
END_VAR

// Safety/GVLs/GPL_Safety
{attribute 'qualified_only'}
{attribute 'global_init_slot' := '40505'}
VAR_GLOBAL CONSTANT
	INDEX_DEVICE_MIN 	: UINT := 1;	
	INDEX_DEVICE_MAX 	: UINT := 1;
	INDEX_GROUP_MIN 	: UINT := 0;	
	INDEX_GROUP_MAX 	: UINT := 3;
END_VAR

// Tests/GC_Test
{attribute 'qualified_only'}
VAR_GLOBAL CONSTANT
	INDEX_TestFB_ActuatorConfigured_MIN			: DINT := 0;
	INDEX_TestFB_ActuatorConfigured_MAX			: DINT := 9;
	INDEX_TestFB_ActuatorInterlock_MIN			: DINT := 0;
	INDEX_TestFB_ActuatorInterlock_MAX			: DINT := 9;
	INDEX_TestFB_BaseStatic_MIN					: DINT := 0;
	INDEX_TestFB_BaseStatic_MAX					: DINT := 1;
	INDEX_TestFB_BaseCyclic_MIN					: DINT := 0;
	INDEX_TestFB_BaseCyclic_MAX					: DINT := 1;
	INDEX_TestFB_Command_MIN					: DINT := 0;
	INDEX_TestFB_Command_MAX					: DINT := 169;
	INDEX_TestFB_Component_MIN					: DINT := 0;
	INDEX_TestFB_Component_MAX					: DINT := 299;
	INDEX_TestFB_PermIntlk_MIN					: DINT := 0;
	INDEX_TestFB_PermIntlk_MAX					: DINT := 299;

	// FB_PermIntlk* Index Allocation Map:
	// ===================================
	// 0-59:   FB_PermIntlkTests - Direct FB_PermIntlk testing
	//         0-9:   Basic functionality tests (existing)
	//         10-19: Transition edge tests (P_OK toggling)
	//         20-29: Idempotence/reinit tests
	//         30-39: Auto-indexing tests for injected configs
	//         40-49: Resolution recovery tests
	//         50-59: Description-driven configured flag tests
	//
	// 60-99:  RESERVED for FB_PermIntlkTests expansion
	//
	// 100-249: FB_CommandTests - FB_PermIntlkCommand instances
	//          NEEDS UPDATE: Many tests currently use indices 6-99 (below 100)
	//          Currently OK: 101,103,200-207 (updated for new runtime tests)
	//          Target range: All TestPermIntlk[x] should use x ∈ [100,249]
	//
	// 250-299: FB_ComponentTests - FB_PermIntlk instances
	//          UPDATED: Extended range to support indices up to 299
	//          Target range: All TestPermIntlk[x] should use x ∈ [250,299]
	//
	// NOTE: FB_ActuatorInterlockTests uses single instance 'fbInterlock' (no array)
	// NOTE: FB_ActuatorConfiguredInterfaceTests uses single 'MockSystemPermIntlk' (no array)
	INDEX_TestFB_FileHandlerCsv_MIN				: DINT := 0;
	INDEX_TestFB_FileHandlerCsv_MAX				: DINT := 9;
	INDEX_TestFB_HashTable_MIN					: DINT := 0;
	INDEX_TestFB_HashTable_MAX					: DINT := 9;
	INDEX_TestFB_RingBuffer_MIN					: DINT := 0;
	INDEX_TestFB_RingBuffer_MAX					: DINT := 61;
	INDEX_TestFB_StringParsing_MIN				: DINT := 0;
	INDEX_TestFB_StringParsing_MAX				: DINT := 2;
	INDEX_TestFB_Sequencer_MIN					: DINT := 0;
	INDEX_TestFB_Sequencer_MAX					: DINT := 39;
	Index_TestFB_Logging_MIN					: DINT := 0;
	Index_TestFB_Logging_MAX					: DINT := 39;
	Index_TestFB_DebounceMIN					: DINT := 0;
	Index_TestFB_DebounceMAX					: DINT := 29;
END_VAR

// Base/POUs/FB_BaseCyclic
FUNCTION_BLOCK ABSTRACT FB_BaseCyclic EXTENDS FB_BaseStatic IMPLEMENTS I_BaseCyclic
VAR
	// Edge-triggered flags for status change logging - prevents log spam
	bLoggedBusyToTrue		: BOOL;
	bLoggedBusyToFalse		: BOOL;
	bLoggedDoneToTrue		: BOOL;
	bLoggedDoneToFalse		: BOOL;
	bLoggedErrorToTrue		: BOOL;
	bLoggedErrorToFalse		: BOOL;
	bLoggedInitializedToTrue	: BOOL;
	bLoggedInitializedToFalse	: BOOL;
	bLoggedEnabledToTrue		: BOOL;
	bLoggedEnabledToFalse		: BOOL;
	bLoggedSimulationToTrue		: BOOL;
	bLoggedSimulationToFalse	: BOOL;
END_VAR

METHOD PROTECTED _ConfigurationCyclic
IF NOT SUPER^.BaseConfiguration.UseLocalConfig THEN
	BaseConfiguration.LogTraceConfiguration.What.xLogToAdsConsole 	:= GPL_Base.xLogToAdsConsole;
	BaseConfiguration.LogTraceConfiguration.What.xLogToEventLogger 	:= GPL_Base.xLogToEventLogger;
	BaseConfiguration.LogTraceConfiguration.What.xLogToFile 		:= GPL_Base.xLogToFile;
	BaseConfiguration.LogTraceConfiguration.When					:= GPL_Base.eLogWhen;
	BaseConfiguration.LogTraceConfiguration.What.MinTraceLevel		:= GPL_Base.PERSISTENT_LOG_LEVEL_MIN;
END_IF
END_METHOD

METHOD PROTECTED _UpdateStatusEdgeTracking
// This method performs edge detection and logging for BaseStatus changes
// Call this at the end of CyclicLogic to detect and log only changes
// Only perform edge detection if verbose tracing is enabled
IF GPL_Base.PERSISTENT_LOG_LEVEL_MIN > Global.TcEventSeverity.Verbose THEN
	RETURN; // Skip edge detection if verbose level is not enabled
END_IF

// Busy edge detection with one-time logging per transition
IF BaseStatus.Busy <> PreviousBaseStatus.Busy THEN
	IF PreviousBaseStatus.Busy THEN
		// Transition: TRUE -> FALSE
		IF NOT bLoggedBusyToFalse THEN
			TraceWithSeverity(Message := 'BaseStatus.Busy: TRUE -> FALSE', Severity := Global.TcEventSeverity.Verbose);
			bLoggedBusyToFalse := TRUE;
		END_IF
		bLoggedBusyToTrue := FALSE; // Reset opposite flag to allow next transition
	ELSE
		// Transition: FALSE -> TRUE
		IF NOT bLoggedBusyToTrue THEN
			TraceWithSeverity(Message := 'BaseStatus.Busy: FALSE -> TRUE', Severity := Global.TcEventSeverity.Verbose);
			bLoggedBusyToTrue := TRUE;
		END_IF
		bLoggedBusyToFalse := FALSE; // Reset opposite flag to allow next transition
	END_IF
	PreviousBaseStatus.Busy := BaseStatus.Busy;
END_IF

// Done edge detection with one-time logging per transition
IF BaseStatus.Done <> PreviousBaseStatus.Done THEN
	IF PreviousBaseStatus.Done THEN
		// Transition: TRUE -> FALSE
		IF NOT bLoggedDoneToFalse THEN
			TraceWithSeverity(Message := 'BaseStatus.Done: TRUE -> FALSE', Severity := Global.TcEventSeverity.Verbose);
			bLoggedDoneToFalse := TRUE;
		END_IF
		bLoggedDoneToTrue := FALSE; // Reset opposite flag to allow next transition
	ELSE
		// Transition: FALSE -> TRUE
		IF NOT bLoggedDoneToTrue THEN
			TraceWithSeverity(Message := 'BaseStatus.Done: FALSE -> TRUE', Severity := Global.TcEventSeverity.Verbose);
			bLoggedDoneToTrue := TRUE;
		END_IF
		bLoggedDoneToFalse := FALSE; // Reset opposite flag to allow next transition
	END_IF
	PreviousBaseStatus.Done := BaseStatus.Done;
END_IF

// Error edge detection with one-time logging per transition
IF BaseStatus.Error <> PreviousBaseStatus.Error THEN
	IF PreviousBaseStatus.Error THEN
		// Transition: TRUE -> FALSE
		IF NOT bLoggedErrorToFalse THEN
			TraceWithSeverity(Message := 'BaseStatus.Error: TRUE -> FALSE', Severity := Global.TcEventSeverity.Verbose);
			bLoggedErrorToFalse := TRUE;
		END_IF
		bLoggedErrorToTrue := FALSE; // Reset opposite flag to allow next transition
	ELSE
		// Transition: FALSE -> TRUE
		IF NOT bLoggedErrorToTrue THEN
			TraceWithSeverity(Message := 'BaseStatus.Error: FALSE -> TRUE', Severity := Global.TcEventSeverity.Verbose);
			bLoggedErrorToTrue := TRUE;
		END_IF
		bLoggedErrorToFalse := FALSE; // Reset opposite flag to allow next transition
	END_IF
	PreviousBaseStatus.Error := BaseStatus.Error;
END_IF

// Initialized edge detection with one-time logging per transition
IF BaseStatus.Initialized <> PreviousBaseStatus.Initialized THEN
	IF PreviousBaseStatus.Initialized THEN
		// Transition: TRUE -> FALSE
		IF NOT bLoggedInitializedToFalse THEN
			TraceWithSeverity(Message := 'BaseStatus.Initialized: TRUE -> FALSE', Severity := Global.TcEventSeverity.Verbose);
			bLoggedInitializedToFalse := TRUE;
		END_IF
		bLoggedInitializedToTrue := FALSE; // Reset opposite flag to allow next transition
	ELSE
		// Transition: FALSE -> TRUE
		IF NOT bLoggedInitializedToTrue THEN
			TraceWithSeverity(Message := 'BaseStatus.Initialized: FALSE -> TRUE', Severity := Global.TcEventSeverity.Verbose);
			bLoggedInitializedToTrue := TRUE;
		END_IF
		bLoggedInitializedToFalse := FALSE; // Reset opposite flag to allow next transition
	END_IF
	PreviousBaseStatus.Initialized := BaseStatus.Initialized;
END_IF

// Enabled edge detection with one-time logging per transition
IF BaseStatus.Enabled <> PreviousBaseStatus.Enabled THEN
	IF PreviousBaseStatus.Enabled THEN
		// Transition: TRUE -> FALSE
		IF NOT bLoggedEnabledToFalse THEN
			TraceWithSeverity(Message := 'BaseStatus.Enabled: TRUE -> FALSE', Severity := Global.TcEventSeverity.Verbose);
			bLoggedEnabledToFalse := TRUE;
		END_IF
		bLoggedEnabledToTrue := FALSE; // Reset opposite flag to allow next transition
	ELSE
		// Transition: FALSE -> TRUE
		IF NOT bLoggedEnabledToTrue THEN
			TraceWithSeverity(Message := 'BaseStatus.Enabled: FALSE -> TRUE', Severity := Global.TcEventSeverity.Verbose);
			bLoggedEnabledToTrue := TRUE;
		END_IF
		bLoggedEnabledToFalse := FALSE; // Reset opposite flag to allow next transition
	END_IF
	PreviousBaseStatus.Enabled := BaseStatus.Enabled;
END_IF

// Simulation edge detection with one-time logging per transition
IF BaseStatus.Simulation <> PreviousBaseStatus.Simulation THEN
	IF PreviousBaseStatus.Simulation THEN
		// Transition: TRUE -> FALSE
		IF NOT bLoggedSimulationToFalse THEN
			TraceWithSeverity(Message := 'BaseStatus.Simulation: TRUE -> FALSE', Severity := Global.TcEventSeverity.Verbose);
			bLoggedSimulationToFalse := TRUE;
		END_IF
		bLoggedSimulationToTrue := FALSE; // Reset opposite flag to allow next transition
	ELSE
		// Transition: FALSE -> TRUE
		IF NOT bLoggedSimulationToTrue THEN
			TraceWithSeverity(Message := 'BaseStatus.Simulation: FALSE -> TRUE', Severity := Global.TcEventSeverity.Verbose);
			bLoggedSimulationToTrue := TRUE;
		END_IF
		bLoggedSimulationToFalse := FALSE; // Reset opposite flag to allow next transition
	END_IF
	PreviousBaseStatus.Simulation := BaseStatus.Simulation;
END_IF
END_METHOD

METHOD CyclicLogic
IF NOT SUPER^.BaseStatus.Initialized THEN
	SUPER^.BaseStatus.Initialized := Initialize();
	RETURN;
END_IF

_ConfigurationCyclic();

// Perform edge detection for BaseStatus changes at end of cycle
_UpdateStatusEdgeTracking();
END_METHOD

PROPERTY Initialized : BOOL
GET
Initialized := SUPER^.BaseStatus.Initialized;
END_GET
END_PROPERTY

END_FUNCTION_BLOCK

// Base/POUs/FB_BaseStatic
{attribute 'reflection'}
FUNCTION_BLOCK ABSTRACT FB_BaseStatic IMPLEMENTS I_BaseStatic
VAR
	BaseConfiguration		: ST_BaseConfiguration;
	BaseStatus				: ST_BaseStatus;
	PreviousBaseStatus		: ST_BaseStatus;

	{attribute 'instance-path'}
	{attribute 'noinit'}
	InstancePath 		: STRING;
END_VAR

PROPERTY Busy : BOOL
GET
Busy := BaseStatus.Busy;
END_GET
END_PROPERTY

PROPERTY Error : BOOL
GET
Error := BaseStatus.Error;
END_GET
END_PROPERTY

PROPERTY ErrorID : UDINT
GET
ErrorID := BaseStatus.ErrorID;
END_GET
END_PROPERTY

METHOD Initialize : BOOL
Initialize	:= _Initialize();
BaseStatus.Initialized := Initialize;
END_METHOD

PROPERTY P_BaseConfiguration : REFERENCE TO ST_BaseConfiguration
GET
P_BaseConfiguration REF= BaseConfiguration;
END_GET
END_PROPERTY

PROPERTY P_BaseStatus : REFERENCE TO ST_BaseStatus
GET
P_BaseStatus REF= BaseStatus;
END_GET
END_PROPERTY

METHOD TraceWithSeverity
VAR_INPUT
	Message		: T_MaxString;
	Severity	: Global.TcEventSeverity;
	RaiseAlarm	: BOOL := FALSE;
END_VAR
// Prevent re-entry to avoid infinite recursion when logging system components call TraceWithSeverity
// Check if already in logging subsystem
IF GVL_System.InReentry_Logging THEN
	RETURN;  // Already in logging subsystem, don't recurse
END_IF

// Check if GVL_System exists
IF NOT __ISVALIDREF(GVL_System.RingBufferLog.P_RingBufferStatus.BaseStatus) THEN
	RETURN;  // No logging system available
END_IF

// All checks passed - now safe to set the re-entry guard
GVL_System.InReentry_Logging := TRUE;

// Check if the logging system exists and is ready
IF __ISVALIDREF(GVL_System.RingBufferLog.P_RingBufferStatus.BaseStatus) THEN
	// If logging system exists but not initialized, try to initialize it
	IF NOT GVL_System.RingBufferLog.P_RingBufferStatus.BaseStatus.Initialized THEN
		GVL_System.RingBufferLog.Initialize();
	END_IF

	// Only log if tracing is enabled and the system is now initialized
	IF GVL_System.RingBufferLog.P_RingBufferStatus.BaseStatus.Initialized AND_THEN GPL_Base.TRACING_ENABLED THEN
		IF Severity >= GPL_Base.PERSISTENT_LOG_LEVEL_MIN THEN
			BaseStatus.LogEntry.Message								:= Message;
			BaseStatus.LogEntry.Severity							:= Severity;
			BaseStatus.LogEntry.RaiseAlarm							:= RaiseAlarm;
			_FormatLogEntry();
			GVL_System.RingBufferLog.AddObject(RefObject := BaseStatus.LogEntry);
		END_IF

		// Verify the entry was added successfully
		IF NOT GVL_System.RingBufferLog.P_ObjectWasAdded THEN
			// AddObject failed - buffer may be full or corrupted
			// Cannot use logging system to report this (would cause recursion)
			// Silently fail - the LogDequeue error handling will detect buffer issues
		ELSE
			// Successfully added - clear the flag
			GVL_System.RingBufferLog.ClearStatusFlagAdded();
		END_IF
	END_IF
END_IF

// Clear re-entry guard before exiting
GVL_System.InReentry_Logging := FALSE;
END_METHOD

METHOD PROTECTED _FormatLogEntry
BaseStatus.LogEntry.InstancePath						:= InstancePath;
BaseStatus.LogEntry.TaskInfo.AdsPort					:= TwinCAT_SystemInfoVarList._TaskInfo[Tc2_System.GETCURTASKINDEXEX()].AdsPort;
BaseStatus.LogEntry.TaskInfo.CycleCount					:= TwinCAT_SystemInfoVarList._TaskInfo[Tc2_System.GETCURTASKINDEXEX()].CycleCount;
BaseStatus.LogEntry.TaskInfo.CycleTime					:= TwinCAT_SystemInfoVarList._TaskInfo[Tc2_System.GETCURTASKINDEXEX()].CycleTime;
BaseStatus.LogEntry.TaskInfo.CycleTimeExceeded			:= TwinCAT_SystemInfoVarList._TaskInfo[Tc2_System.GETCURTASKINDEXEX()].CycleTimeExceeded;
BaseStatus.LogEntry.TaskInfo.DcTaskTime					:= TwinCAT_SystemInfoVarList._TaskInfo[Tc2_System.GETCURTASKINDEXEX()].DcTaskTime;
BaseStatus.LogEntry.TaskInfo.FirstCycle					:= TwinCAT_SystemInfoVarList._TaskInfo[Tc2_System.GETCURTASKINDEXEX()].FirstCycle;
//		BaseStatus.LogEntry.TaskInfo.InCallAfterOutputUpdate	:= TwinCAT_SystemInfoVarList._TaskInfo[Tc2_System.GETCURTASKINDEXEX()].InCallAfterOutputUpdate;
BaseStatus.LogEntry.TaskInfo.LastExecTime				:= TwinCAT_SystemInfoVarList._TaskInfo[Tc2_System.GETCURTASKINDEXEX()].LastExecTime;
BaseStatus.LogEntry.TaskInfo.ObjId						:= TwinCAT_SystemInfoVarList._TaskInfo[Tc2_System.GETCURTASKINDEXEX()].ObjId;
BaseStatus.LogEntry.TaskInfo.Priority					:= TwinCAT_SystemInfoVarList._TaskInfo[Tc2_System.GETCURTASKINDEXEX()].Priority;
BaseStatus.LogEntry.TaskInfo.RTViolation				:= TwinCAT_SystemInfoVarList._TaskInfo[Tc2_System.GETCURTASKINDEXEX()].RTViolation;
BaseStatus.LogEntry.TaskInfo.TaskName					:= TwinCAT_SystemInfoVarList._TaskInfo[Tc2_System.GETCURTASKINDEXEX()].TaskName;
END_METHOD

// Basic component initialization logic
METHOD PROTECTED _Initialize : BOOL;
// This method is called by CyclicLogic() as required
VAR
	InterimInit : BOOL;
END_VAR
// Initialize children dependencies first
InterimInit := _InitializeChildrenDependencies();
IF NOT InterimInit THEN
	IF BaseConfiguration.LogTraceConfiguration.What.xLogToEventLogger AND NOT BaseStatus.LogTraceStatus.InitChildrenFailureShown THEN
		TraceWithSeverity(Message := Tc2_Standard.CONCAT('_InitializeChildrenDependencies Failed at ', __POUNAME()), Severity := Global.TcEventSeverity.Error);
		BaseStatus.LogTraceStatus.InitChildrenFailureShown := TRUE;
	END_IF
	_Initialize := FALSE;
	RETURN;
END_IF

// Initialize references second
InterimInit := _InitializeReferences();
IF NOT InterimInit THEN
	IF BaseConfiguration.LogTraceConfiguration.What.xLogToEventLogger AND NOT BaseStatus.LogTraceStatus.InitReferencesFailureShown THEN
		TraceWithSeverity(Message := Tc2_Standard.CONCAT('_InitializeReferences Failed at ', __POUNAME()), Severity := Global.TcEventSeverity.Error);
		BaseStatus.LogTraceStatus.InitReferencesFailureShown := TRUE;
	END_IF
	_Initialize := FALSE;
	RETURN;
END_IF

// Set dependency configuration last
InterimInit := _SetDependencyConfiguration();
IF NOT InterimInit THEN
	IF BaseConfiguration.LogTraceConfiguration.What.xLogToEventLogger AND NOT BaseStatus.LogTraceStatus.InitDependencyConfigFailureShown THEN
		TraceWithSeverity(Message := Tc2_Standard.CONCAT('_SetDependencyConfiguration Failed at ', __POUNAME()), Severity := Global.TcEventSeverity.Error);
		BaseStatus.LogTraceStatus.InitDependencyConfigFailureShown := TRUE;
	END_IF
	_Initialize := FALSE;
	RETURN;
END_IF

// All initialization steps succeeded
_Initialize := TRUE;
END_METHOD

{warning 'Initialization may have failed.  Have you overwritten this method with your final implementation?'}
{warning 'Do not call again - already called in FB_Base'}
METHOD PROTECTED _InitializeChildrenDependencies : BOOL
_InitializeChildrenDependencies := TRUE;
END_METHOD

METHOD PROTECTED _InitializeReferences : BOOL
//Order is important!
BaseConfiguration.InstancePath 	REF= InstancePath;

// Show initialization message only once per instance, not on every retry
IF NOT BaseStatus.LogTraceStatus.MessageShown AND
   BaseConfiguration.LogTraceConfiguration.When = E_LogTraceWhen.xRunOnInitOnly AND_THEN
   BaseConfiguration.LogTraceConfiguration.What.xLogToEventLogger THEN
	TraceWithSeverity(Message := Tc2_Standard.CONCAT('If you created new data structures, they may not have valid pointer references; Check ', __POUNAME()), Severity := Global.TcEventSeverity.Warning);
	BaseStatus.LogTraceStatus.MessageShown := TRUE;
END_IF

_InitializeReferences 			:= TRUE; // apply at end of all reference initialization
END_METHOD

METHOD PROTECTED _SetDependencyConfiguration : BOOL
_SetDependencyConfiguration	:= TRUE;
END_METHOD

METHOD RaiseAlarm
VAR_INPUT
	Message		: T_MaxString;
	Severity	: Global.TcEventSeverity;
	RaiseAlarm	: BOOL := TRUE;
END_VAR
// Prevent re-entry to avoid infinite recursion when logging system components call RaiseAlarm
// Check if already in logging subsystem
IF GVL_System.InReentry_Logging THEN
	RETURN;  // Already in logging subsystem, don't recurse
END_IF

// Check if GVL_System exists
IF NOT __ISVALIDREF(GVL_System.RingBufferLog.P_RingBufferStatus.BaseStatus) THEN
	RETURN;  // No logging system available
END_IF

// All checks passed - now safe to set the re-entry guard
GVL_System.InReentry_Logging := TRUE;

// Check if the logging system exists and is ready
IF __ISVALIDREF(GVL_System.RingBufferLog.P_RingBufferStatus.BaseStatus) THEN
	// If logging system exists but not initialized, try to initialize it
	IF NOT GVL_System.RingBufferLog.P_RingBufferStatus.BaseStatus.Initialized THEN
		GVL_System.RingBufferLog.Initialize();
	END_IF

